LIN {X 0,Y 679.912,Z 1280.609,A -85,B 0,C 180,E1 32312.866,E2 32312.866} C_VEL
LIN {X 0,Y 679.874,Z 1281.737,A -85,B 0,C 180,E1 32311.011,E2 32311.011} C_VEL
LIN {X 0,Y 679.863,Z 1281.827,A -85,B 0,C 180,E1 32309.326,E2 32309.326} C_VEL
LIN {X 0,Y 679.905,Z 1280.946,A -85,B 0,C 180,E1 32307.556,E2 32307.556} C_VEL
LIN {X 0,Y 679.915,Z 1278.919,A -85,B 0,C 180,E1 32305.614,E2 32305.614} C_VEL
LIN {X 0,Y 679.929,Z 1274.906,A -85,B 0,C 180,E1 32303.329,E2 32303.329} C_VEL
LIN {X 0,Y 679.943,Z 1269.331,A -85,B 0,C 180,E1 32301.118,E2 32301.118} C_VEL
LIN {X 0,Y 680.017,Z 1263.356,A -85,B 0,C 180,E1 32299.238,E2 32299.238} C_VEL
LIN {X 0,Y 680.138,Z 1256.508,A -85,B 0,C 180,E1 32297.433,E2 32297.433} C_VEL
LIN {X 0,Y 680.303,Z 1248.399,A -85,B 0,C 180,E1 32295.6,E2 32295.6} C_VEL
LIN {X 0,Y 680.525,Z 1238.351,A -85,B 0,C 180,E1 32293.628,E2 32293.628} C_VEL
LIN {X 0,Y 680.966,Z 1224.744,A -85,B 0,C 180,E1 32291.331,E2 32291.331} C_VEL
LIN {X 0,Y 681.406,Z 1211.769,A -85,B 0,C 180,E1 32289.423,E2 32289.423} C_VEL
LIN {X 0,Y 681.969,Z 1198.553,A -85,B 0,C 180,E1 32287.683,E2 32287.683} C_VEL
LIN {X 0,Y 682.78,Z 1180.927,A -85,B 0,C 180,E1 32285.609,E2 32285.609} C_VEL
LIN {X 0,Y 683.632,Z 1163.822,A -85,B 0,C 180,E1 32283.831,E2 32283.831} C_VEL
LIN {X 0,Y 684.499,Z 1146.752,A -85,B 0,C 180,E1 32282.227,E2 32282.227} C_VEL
LIN {X 0,Y 685.785,Z 1124.203,A -85,B 0,C 180,E1 32280.341,E2 32280.341} C_VEL
LIN {X 0,Y 686.866,Z 1105.235,A -85,B 0,C 180,E1 32278.932,E2 32278.932} C_VEL
LIN {X 0,Y 687.97,Z 1085.493,A -85,B 0,C 180,E1 32277.61,E2 32277.61} C_VEL
LIN {X 0,Y 689.441,Z 1059.992,A -85,B 0,C 180,E1 32276.108,E2 32276.108} C_VEL
LIN {X 0,Y 690.593,Z 1038.701,A -85,B 0,C 180,E1 32275.016,E2 32275.016} C_VEL
LIN {X 0,Y 691.622,Z 1018.737,A -85,B 0,C 180,E1 32274.11,E2 32274.11} C_VEL
LIN {X 0,Y 692.593,Z 998.313,A -85,B 0,C 180,E1 32273.296,E2 32273.296} C_VEL
LIN {X 0,Y 693.528,Z 975.949,A -85,B 0,C 180,E1 32272.526,E2 32272.526} C_VEL
LIN {X 0,Y 694.563,Z 949.849,A -85,B 0,C 180,E1 32271.785,E2 32271.785} C_VEL
LIN {X 0,Y 695.355,Z 923.524,A -85,B 0,C 180,E1 32271.209,E2 32271.209} C_VEL
LIN {X 0,Y 695.921,Z 898.887,A -85,B 0,C 180,E1 32270.809,E2 32270.809} C_VEL
LIN {X 0,Y 698.303,Z 673.986,A -85,B 0,C 180,E1 32267.976,E2 32267.976} C_VEL
LIN {X 0,Y 700.559,Z 471.336,A -85,B 0,C 180,E1 32265.348,E2 32265.348} C_VEL
LIN {X 0,Y 700.664,Z 446.208,A -85,B 0,C 180,E1 32265,E2 32265} C_VEL
LIN {X 0,Y 696.356,Z 426.818,A -85,B 0,C 180,E1 32264.352,E2 32264.352} C_VEL
LIN {X 0,Y 698.129,Z 385.1,A -85,B 0,C 180,E1 32261.709,E2 32261.709} C_VEL
LIN {X 0,Y 698.689,Z 371.907,A -85,B 0,C 180,E1 32260.845,E2 32260.845} C_VEL
LIN {X 0,Y 684.161,Z 344.352,A -85,B 0,C 180,E1 32257.655,E2 32257.655} C_VEL
LIN {X 0,Y 682.069,Z 340.229,A -85,B 0,C 180,E1 32257.156,E2 32257.156} C_VEL
LIN {X 0,Y 680.532,Z 336.669,A -85,B 0,C 180,E1 32256.697,E2 32256.697} C_VEL
LIN {X 0,Y 680.502,Z 336.461,A -85,B 0,C 180,E1 32254.78,E2 32254.78} C_VEL
LIN {X 0,Y 680.517,Z 336.464,A -85,B 0,C 180,E1 32251.836,E2 32251.836} C_VEL
LIN {X 0,Y 680.507,Z 336.459,A -85,B 0,C 180,E1 32248.812,E2 32248.812} C_VEL
LIN {X 0,Y 680.521,Z 336.455,A -85,B 0,C 180,E1 32245.754,E2 32245.754} C_VEL
LIN {X 0,Y 680.506,Z 336.467,A -85,B 0,C 180,E1 32242.642,E2 32242.642} C_VEL
LIN {X 0,Y 680.523,Z 336.458,A -85,B 0,C 180,E1 32239.573,E2 32239.573} C_VEL
LIN {X 0,Y 680.505,Z 336.464,A -85,B 0,C 180,E1 32236.474,E2 32236.474} C_VEL
LIN {X 0,Y 680.526,Z 336.457,A -85,B 0,C 180,E1 32233.424,E2 32233.424} C_VEL
LIN {X 0,Y 680.505,Z 336.465,A -85,B 0,C 180,E1 32230.327,E2 32230.327} C_VEL
LIN {X 0,Y 680.526,Z 336.455,A -85,B 0,C 180,E1 32227.259,E2 32227.259} C_VEL
LIN {X 0,Y 680.502,Z 336.466,A -85,B 0,C 180,E1 32224.129,E2 32224.129} C_VEL
LIN {X 0,Y 680.518,Z 336.451,A -85,B 0,C 180,E1 32221.094,E2 32221.094} C_VEL
LIN {X 0,Y 680.501,Z 336.465,A -85,B 0,C 180,E1 32217.979,E2 32217.979} C_VEL
LIN {X 0,Y 680.509,Z 336.456,A -85,B 0,C 180,E1 32214.996,E2 32214.996} C_VEL
LIN {X 0,Y 680.499,Z 336.465,A -85,B 0,C 180,E1 32211.806,E2 32211.806} C_VEL
LIN {X 0,Y 680.497,Z 336.458,A -85,B 0,C 180,E1 32208.902,E2 32208.902} C_VEL
LIN {X 0,Y 680.505,Z 336.465,A -85,B 0,C 180,E1 32205.709,E2 32205.709} C_VEL
LIN {X 0,Y 680.486,Z 336.455,A -85,B 0,C 180,E1 32202.822,E2 32202.822} C_VEL
LIN {X 0,Y 680.522,Z 336.462,A -85,B 0,C 180,E1 32199.711,E2 32199.711} C_VEL
LIN {X 0,Y 680.475,Z 336.457,A -85,B 0,C 180,E1 32196.809,E2 32196.809} C_VEL
LIN {X 0,Y 680.527,Z 336.461,A -85,B 0,C 180,E1 32193.846,E2 32193.846} C_VEL
LIN {X 0,Y 680.473,Z 336.459,A -85,B 0,C 180,E1 32190.897,E2 32190.897} C_VEL
LIN {X 0,Y 680.524,Z 336.463,A -85,B 0,C 180,E1 32189.443,E2 32189.443} C_VEL
LIN {X 0,Y 679.498,Z 336.6,A -85,B 0,C 180,E1 32188.795,E2 32188.795} C_VEL
LIN {X 0,Y 673.053,Z 337.39,A -85,B 0,C 180,E1 32186.977,E2 32186.977} C_VEL
LIN {X 0,Y 672.532,Z 337.45,A -85,B 0,C 180,E1 32186.504,E2 32186.504} C_VEL
LIN {X 0,Y 672.587,Z 337.447,A -85,B 0,C 180,E1 32183.512,E2 32183.512} C_VEL
LIN {X 0,Y 672.53,Z 337.452,A -85,B 0,C 180,E1 32180.591,E2 32180.591} C_VEL
LIN {X 0,Y 672.563,Z 337.445,A -85,B 0,C 180,E1 32177.762,E2 32177.762} C_VEL
LIN {X 0,Y 672.544,Z 337.454,A -85,B 0,C 180,E1 32174.685,E2 32174.685} C_VEL
LIN {X 0,Y 672.526,Z 337.448,A -85,B 0,C 180,E1 32171.979,E2 32171.979} C_VEL
LIN {X 0,Y 672.59,Z 337.451,A -85,B 0,C 180,E1 32168.964,E2 32168.964} C_VEL
LIN {X 0,Y 672.519,Z 337.45,A -85,B 0,C 180,E1 32166.069,E2 32166.069} C_VEL
LIN {X 0,Y 672.562,Z 337.45,A -85,B 0,C 180,E1 32163.27,E2 32163.27} C_VEL
LIN {X 0,Y 672.53,Z 337.451,A -85,B 0,C 180,E1 32160.167,E2 32160.167} C_VEL
LIN {X 0,Y 672.519,Z 337.451,A -85,B 0,C 180,E1 32157.541,E2 32157.541} C_VEL
LIN {X 0,Y 672.585,Z 337.452,A -85,B 0,C 180,E1 32154.505,E2 32154.505} C_VEL
LIN {X 0,Y 672.512,Z 337.453,A -85,B 0,C 180,E1 32151.637,E2 32151.637} C_VEL
LIN {X 0,Y 672.545,Z 337.452,A -85,B 0,C 180,E1 32148.911,E2 32148.911} C_VEL
LIN {X 0,Y 672.525,Z 337.452,A -85,B 0,C 180,E1 32145.788,E2 32145.788} C_VEL
LIN {X 0,Y 672.505,Z 337.454,A -85,B 0,C 180,E1 32143.236,E2 32143.236} C_VEL
LIN {X 0,Y 672.566,Z 337.453,A -85,B 0,C 180,E1 32140.45,E2 32140.45} C_VEL
LIN {X 0,Y 672.511,Z 337.455,A -85,B 0,C 180,E1 32137.432,E2 32137.432} C_VEL
LIN {X 0,Y 672.501,Z 337.451,A -85,B 0,C 180,E1 32134.947,E2 32134.947} C_VEL
LIN {X 0,Y 672.58,Z 337.45,A -85,B 0,C 180,E1 32132.045,E2 32132.045} C_VEL
LIN {X 0,Y 672.505,Z 337.457,A -85,B 0,C 180,E1 32129.148,E2 32129.148} C_VEL
LIN {X 0,Y 672.498,Z 337.444,A -85,B 0,C 180,E1 32126.591,E2 32126.591} C_VEL
LIN {X 0,Y 672.576,Z 337.438,A -85,B 0,C 180,E1 32123.598,E2 32123.598} C_VEL
LIN {X 0,Y 672.493,Z 337.458,A -85,B 0,C 180,E1 32120.76,E2 32120.76} C_VEL
LIN {X 0,Y 672.498,Z 337.454,A -85,B 0,C 180,E1 32118.247,E2 32118.247} C_VEL
LIN {X 0,Y 672.554,Z 337.396,A -85,B 0,C 180,E1 32115.273,E2 32115.273} C_VEL
LIN {X 0,Y 672.486,Z 337.444,A -85,B 0,C 180,E1 32112.522,E2 32112.522} C_VEL
LIN {X 0,Y 672.557,Z 337.781,A -85,B 0,C 180,E1 32111.853,E2 32111.853} C_VEL
LIN {X 0,Y 673.067,Z 339.501,A -85,B 0,C 180,E1 32111.692,E2 32111.692} C_VEL
LIN {X 0,Y 675.158,Z 342.401,A -85,B 0,C 180,E1 32111.458,E2 32111.458} C_VEL
LIN {X 0,Y 676.417,Z 343.843,A -85,B 0,C 180,E1 32111.324,E2 32111.324} C_VEL
LIN {X 0,Y 679.051,Z 347.701,A -85,B 0,C 180,E1 32111.034,E2 32111.034} C_VEL
LIN {X 0,Y 690.723,Z 363.983,A -85,B 0,C 180,E1 32109.803,E2 32109.803} C_VEL
LIN {X 0,Y 694.272,Z 369.404,A -85,B 0,C 180,E1 32109.435,E2 32109.435} C_VEL
LIN {X 0,Y 691.631,Z 585.542,A -85,B 0,C 180,E1 32106.635,E2 32106.635} C_VEL
LIN {X 0,Y 689.568,Z 757.13,A -85,B 0,C 180,E1 32104.45,E2 32104.45} C_VEL
LIN {X 0,Y 688.782,Z 783.452,A -85,B 0,C 180,E1 32103.968,E2 32103.968} C_VEL
LIN {X 0,Y 687.772,Z 810.9,A -85,B 0,C 180,E1 32103.292,E2 32103.292} C_VEL
LIN {X 0,Y 686.614,Z 836.969,A -85,B 0,C 180,E1 32102.482,E2 32102.482} C_VEL
LIN {X 0,Y 685.243,Z 863.991,A -85,B 0,C 180,E1 32101.454,E2 32101.454} C_VEL
LIN {X 0,Y 683.973,Z 886.619,A -85,B 0,C 180,E1 32100.439,E2 32100.439} C_VEL
LIN {X 0,Y 682.54,Z 910.71,A -85,B 0,C 180,E1 32099.198,E2 32099.198} C_VEL
LIN {X 0,Y 680.907,Z 936.023,A -85,B 0,C 180,E1 32097.689,E2 32097.689} C_VEL
LIN {X 0,Y 679.643,Z 956.28,A -85,B 0,C 180,E1 32096.315,E2 32096.315} C_VEL
LIN {X 0,Y 678.282,Z 978.203,A -85,B 0,C 180,E1 32094.648,E2 32094.648} C_VEL
LIN {X 0,Y 676.938,Z 999.251,A -85,B 0,C 180,E1 32092.835,E2 32092.835} C_VEL
LIN {X 0,Y 675.887,Z 1017.79,A -85,B 0,C 180,E1 32091.044,E2 32091.044} C_VEL
LIN {X 0,Y 674.833,Z 1036.227,A -85,B 0,C 180,E1 32089.037,E2 32089.037} C_VEL
LIN {X 0,Y 674.017,Z 1053.07,A -85,B 0,C 180,E1 32086.969,E2 32086.969} C_VEL
LIN {X 0,Y 673.315,Z 1068.958,A -85,B 0,C 180,E1 32084.741,E2 32084.741} C_VEL
LIN {X 0,Y 672.867,Z 1081.301,A -85,B 0,C 180,E1 32082.771,E2 32082.771} C_VEL
LIN {X 0,Y 672.493,Z 1093.06,A -85,B 0,C 180,E1 32080.635,E2 32080.635} C_VEL
LIN {X 0,Y 672.222,Z 1104.249,A -85,B 0,C 180,E1 32078.227,E2 32078.227} C_VEL
LIN {X 0,Y 672.062,Z 1112.122,A -85,B 0,C 180,E1 32076.204,E2 32076.204} C_VEL
LIN {X 0,Y 671.984,Z 1118.828,A -85,B 0,C 180,E1 32074.123,E2 32074.123} C_VEL
LIN {X 0,Y 671.93,Z 1124.669,A -85,B 0,C 180,E1 32071.823,E2 32071.823} C_VEL
LIN {X 0,Y 671.911,Z 1128.607,A -85,B 0,C 180,E1 32069.608,E2 32069.608} C_VEL
LIN {X 0,Y 671.882,Z 1130.912,A -85,B 0,C 180,E1 32067.508,E2 32067.508} C_VEL
LIN {X 0,Y 671.901,Z 1131.864,A -85,B 0,C 180,E1 32065.567,E2 32065.567} C_VEL
LIN {X 0,Y 671.887,Z 1131.578,A -85,B 0,C 180,E1 32063.32,E2 32063.32} C_VEL
LIN {X 0,Y 671.909,Z 1129.575,A -85,B 0,C 180,E1 32061.017,E2 32061.017} C_VEL
LIN {X 0,Y 671.92,Z 1126.17,A -85,B 0,C 180,E1 32058.84,E2 32058.84} C_VEL
LIN {X 0,Y 671.953,Z 1120.892,A -85,B 0,C 180,E1 32056.512,E2 32056.512} C_VEL
LIN {X 0,Y 671.997,Z 1113.905,A -85,B 0,C 180,E1 32054.212,E2 32054.212} C_VEL
LIN {X 0,Y 672.161,Z 1106.347,A -85,B 0,C 180,E1 32052.195,E2 32052.195} C_VEL
LIN {X 0,Y 672.346,Z 1097.951,A -85,B 0,C 180,E1 32050.28,E2 32050.28} C_VEL
LIN {X 0,Y 672.66,Z 1086.935,A -85,B 0,C 180,E1 32048.118,E2 32048.118} C_VEL
LIN {X 0,Y 673.123,Z 1073.623,A -85,B 0,C 180,E1 32045.883,E2 32045.883} C_VEL
LIN {X 0,Y 673.696,Z 1060.257,A -85,B 0,C 180,E1 32043.915,E2 32043.915} C_VEL
LIN {X 0,Y 674.445,Z 1044.62,A -85,B 0,C 180,E1 32041.869,E2 32041.869} C_VEL
LIN {X 0,Y 675.363,Z 1026.896,A -85,B 0,C 180,E1 32039.83,E2 32039.83} C_VEL
LIN {X 0,Y 676.458,Z 1007.895,A -85,B 0,C 180,E1 32037.882,E2 32037.882} C_VEL
LIN {X 0,Y 677.675,Z 987.343,A -85,B 0,C 180,E1 32036.024,E2 32036.024} C_VEL
LIN {X 0,Y 678.875,Z 968.036,A -85,B 0,C 180,E1 32034.464,E2 32034.464} C_VEL
LIN {X 0,Y 680.414,Z 944.599,A -85,B 0,C 180,E1 32032.782,E2 32032.782} C_VEL
LIN {X 0,Y 681.858,Z 921.205,A -85,B 0,C 180,E1 32031.313,E2 32031.313} C_VEL
LIN {X 0,Y 683.375,Z 896.661,A -85,B 0,C 180,E1 32029.962,E2 32029.962} C_VEL
LIN {X 0,Y 684.813,Z 872.081,A -85,B 0,C 180,E1 32028.802,E2 32028.802} C_VEL
LIN {X 0,Y 686.072,Z 848.377,A -85,B 0,C 180,E1 32027.843,E2 32027.843} C_VEL
LIN {X 0,Y 687.209,Z 824.159,A -85,B 0,C 180,E1 32027.009,E2 32027.009} C_VEL
LIN {X 0,Y 688.249,Z 798.684,A -85,B 0,C 180,E1 32026.296,E2 32026.296} C_VEL
LIN {X 0,Y 689.148,Z 771.844,A -85,B 0,C 180,E1 32025.71,E2 32025.71} C_VEL
LIN {X 0,Y 689.804,Z 745.156,A -85,B 0,C 180,E1 32025.292,E2 32025.292} C_VEL
LIN {X 0,Y 692.457,Z 516.247,A -85,B 0,C 180,E1 32022.387,E2 32022.387} C_VEL
LIN {X 0,Y 694.14,Z 368.783,A -85,B 0,C 180,E1 32020.455,E2 32020.455} C_VEL
LIN {X 0,Y 682.65,Z 352.629,A -85,B 0,C 180,E1 32019.262,E2 32019.262} C_VEL
LIN {X 0,Y 678.852,Z 347.456,A -85,B 0,C 180,E1 32018.855,E2 32018.855} C_VEL
LIN {X 0,Y 676.214,Z 343.332,A -85,B 0,C 180,E1 32018.56,E2 32018.56} C_VEL
LIN {X 0,Y 673.433,Z 340.156,A -85,B 0,C 180,E1 32018.263,E2 32018.263} C_VEL
LIN {X 0,Y 672.641,Z 337.945,A -85,B 0,C 180,E1 32018.092,E2 32018.092} C_VEL
LIN {X 0,Y 672.533,Z 337.461,A -85,B 0,C 180,E1 32017.721,E2 32017.721} C_VEL
LIN {X 0,Y 672.565,Z 337.457,A -85,B 0,C 180,E1 32014.874,E2 32014.874} C_VEL
LIN {X 0,Y 672.558,Z 337.453,A -85,B 0,C 180,E1 32011.786,E2 32011.786} C_VEL
LIN {X 0,Y 672.567,Z 337.457,A -85,B 0,C 180,E1 32008.844,E2 32008.844} C_VEL
LIN {X 0,Y 672.574,Z 337.453,A -85,B 0,C 180,E1 32005.705,E2 32005.705} C_VEL
LIN {X 0,Y 672.609,Z 337.669,A -85,B 0,C 180,E1 32002.684,E2 32002.684} C_VEL
LIN {X 0,Y 673.551,Z 340.405,A -85,B 0,C 180,E1 32002.401,E2 32002.401} C_VEL
LIN {X 0,Y 681.915,Z 359.556,A -85,B 0,C 180,E1 32000.804,E2 32000.804} C_VEL
LIN {X 0,Y 692.135,Z 376.102,A -85,B 0,C 180,E1 31999.37,E2 31999.37} C_VEL
LIN {X 0,Y 692.068,Z 388.415,A -85,B 0,C 180,E1 31998.624,E2 31998.624} C_VEL
LIN {X 0,Y 690.346,Z 427.413,A -85,B 0,C 180,E1 31996.143,E2 31996.143} C_VEL
LIN {X 0,Y 695.134,Z 449.846,A -85,B 0,C 180,E1 31995.405,E2 31995.405} C_VEL
LIN {X 0,Y 692.574,Z 656.228,A -85,B 0,C 180,E1 31992.697,E2 31992.697} C_VEL
LIN {X 0,Y 689.978,Z 881.138,A -85,B 0,C 180,E1 31989.841,E2 31989.841} C_VEL
LIN {X 0,Y 689.357,Z 915.017,A -85,B 0,C 180,E1 31989.367,E2 31989.367} C_VEL
LIN {X 0,Y 688.525,Z 940.749,A -85,B 0,C 180,E1 31988.848,E2 31988.848} C_VEL
LIN {X 0,Y 687.58,Z 965.293,A -85,B 0,C 180,E1 31988.212,E2 31988.212} C_VEL
LIN {X 0,Y 686.32,Z 993.267,A -85,B 0,C 180,E1 31987.301,E2 31987.301} C_VEL
LIN {X 0,Y 685.156,Z 1015.348,A -85,B 0,C 180,E1 31986.438,E2 31986.438} C_VEL
LIN {X 0,Y 684.01,Z 1035.71,A -85,B 0,C 180,E1 31985.525,E2 31985.525} C_VEL
LIN {X 0,Y 682.83,Z 1055.546,A -85,B 0,C 180,E1 31984.52,E2 31984.52} C_VEL
LIN {X 0,Y 681.501,Z 1077.263,A -85,B 0,C 180,E1 31983.279,E2 31983.279} C_VEL
LIN {X 0,Y 679.886,Z 1101.91,A -85,B 0,C 180,E1 31981.67,E2 31981.67} C_VEL
LIN {X 0,Y 678.73,Z 1120.318,A -85,B 0,C 180,E1 31980.312,E2 31980.312} C_VEL
LIN {X 0,Y 677.63,Z 1138.267,A -85,B 0,C 180,E1 31978.849,E2 31978.849} C_VEL
LIN {X 0,Y 676.325,Z 1159.658,A -85,B 0,C 180,E1 31976.897,E2 31976.897} C_VEL
LIN {X 0,Y 675.387,Z 1175.867,A -85,B 0,C 180,E1 31975.234,E2 31975.234} C_VEL
LIN {X 0,Y 674.605,Z 1191.175,A -85,B 0,C 180,E1 31973.497,E2 31973.497} C_VEL
LIN {X 0,Y 673.761,Z 1208.709,A -85,B 0,C 180,E1 31971.254,E2 31971.254} C_VEL
LIN {X 0,Y 673.218,Z 1221.848,A -85,B 0,C 180,E1 31969.342,E2 31969.342} C_VEL
LIN {X 0,Y 672.774,Z 1233.631,A -85,B 0,C 180,E1 31967.416,E2 31967.416} C_VEL
LIN {X 0,Y 672.399,Z 1246.43,A -85,B 0,C 180,E1 31964.995,E2 31964.995} C_VEL
LIN {X 0,Y 672.194,Z 1255.439,A -85,B 0,C 180,E1 31962.98,E2 31962.98} C_VEL
LIN {X 0,Y 672.049,Z 1262.44,A -85,B 0,C 180,E1 31961.152,E2 31961.152} C_VEL
LIN {X 0,Y 671.943,Z 1268.053,A -85,B 0,C 180,E1 31959.421,E2 31959.421} C_VEL
LIN {X 0,Y 671.921,Z 1273.165,A -85,B 0,C 180,E1 31957.525,E2 31957.525} C_VEL
LIN {X 0,Y 671.914,Z 1277.634,A -85,B 0,C 180,E1 31955.294,E2 31955.294} C_VEL
LIN {X 0,Y 671.909,Z 1280.473,A -85,B 0,C 180,E1 31953.071,E2 31953.071} C_VEL
LIN {X 0,Y 671.881,Z 1281.715,A -85,B 0,C 180,E1 31951.108,E2 31951.108} C_VEL
LIN {X 0,Y 671.863,Z 1281.827,A -85,B 0,C 180,E1 31949.318,E2 31949.318} C_VEL
LIN {X 0,Y 671.906,Z 1280.946,A -85,B 0,C 180,E1 31947.527,E2 31947.527} C_VEL
LIN {X 0,Y 671.913,Z 1278.916,A -85,B 0,C 180,E1 31945.562,E2 31945.562} C_VEL
LIN {X 0,Y 671.928,Z 1274.907,A -85,B 0,C 180,E1 31943.249,E2 31943.249} C_VEL
LIN {X 0,Y 671.947,Z 1269.585,A -85,B 0,C 180,E1 31941.097,E2 31941.097} C_VEL
LIN {X 0,Y 672.032,Z 1263.357,A -85,B 0,C 180,E1 31939.108,E2 31939.108} C_VEL
LIN {X 0,Y 672.175,Z 1256.509,A -85,B 0,C 180,E1 31937.282,E2 31937.282} C_VEL
LIN {X 0,Y 672.367,Z 1248.072,A -85,B 0,C 180,E1 31935.356,E2 31935.356} C_VEL
LIN {X 0,Y 672.673,Z 1236.883,A -85,B 0,C 180,E1 31933.151,E2 31933.151} C_VEL
LIN {X 0,Y 673.15,Z 1223.595,A -85,B 0,C 180,E1 31930.926,E2 31930.926} C_VEL
LIN {X 0,Y 673.654,Z 1210.816,A -85,B 0,C 180,E1 31929.041,E2 31929.041} C_VEL
LIN {X 0,Y 674.368,Z 1195.631,A -85,B 0,C 180,E1 31927.038,E2 31927.038} C_VEL
LIN {X 0,Y 675.303,Z 1177.849,A -85,B 0,C 180,E1 31924.981,E2 31924.981} C_VEL
LIN {X 0,Y 676.174,Z 1161.986,A -85,B 0,C 180,E1 31923.334,E2 31923.334} C_VEL
LIN {X 0,Y 677.396,Z 1142.684,A -85,B 0,C 180,E1 31921.526,E2 31921.526} C_VEL
LIN {X 0,Y 678.65,Z 1121.656,A -85,B 0,C 180,E1 31919.792,E2 31919.792} C_VEL
LIN {X 0,Y 679.836,Z 1102.674,A -85,B 0,C 180,E1 31918.385,E2 31918.385} C_VEL
LIN {X 0,Y 681.412,Z 1078.863,A -85,B 0,C 180,E1 31916.816,E2 31916.816} C_VEL
LIN {X 0,Y 682.768,Z 1056.609,A -85,B 0,C 180,E1 31915.538,E2 31915.538} C_VEL
LIN {X 0,Y 683.963,Z 1036.588,A -85,B 0,C 180,E1 31914.517,E2 31914.517} C_VEL
LIN {X 0,Y 685.098,Z 1016.48,A -85,B 0,C 180,E1 31913.61,E2 31913.61} C_VEL
LIN {X 0,Y 686.225,Z 995.033,A -85,B 0,C 180,E1 31912.765,E2 31912.765} C_VEL
LIN {X 0,Y 687.499,Z 967.39,A -85,B 0,C 180,E1 31911.848,E2 31911.848} C_VEL
LIN {X 0,Y 688.481,Z 941.923,A -85,B 0,C 180,E1 31911.179,E2 31911.179} C_VEL
LIN {X 0,Y 689.293,Z 917.142,A -85,B 0,C 180,E1 31910.671,E2 31910.671} C_VEL
LIN {X 0,Y 689.928,Z 885.559,A -85,B 0,C 180,E1 31910.215,E2 31910.215} C_VEL
LIN {X 0,Y 692.512,Z 661.135,A -85,B 0,C 180,E1 31907.366,E2 31907.366} C_VEL
LIN {X 0,Y 695.041,Z 456.954,A -85,B 0,C 180,E1 31904.69,E2 31904.69} C_VEL
LIN {X 0,Y 694.977,Z 448.325,A -85,B 0,C 180,E1 31904.56,E2 31904.56} C_VEL
LIN {X 0,Y 690.269,Z 426.618,A -85,B 0,C 180,E1 31903.821,E2 31903.821} C_VEL
LIN {X 0,Y 692.248,Z 383.567,A -85,B 0,C 180,E1 31901.064,E2 31901.064} C_VEL
LIN {X 0,Y 692.335,Z 376.179,A -85,B 0,C 180,E1 31900.584,E2 31900.584} C_VEL
LIN {X 0,Y 678.51,Z 349.688,A -85,B 0,C 180,E1 31897.49,E2 31897.49} C_VEL
LIN {X 0,Y 676.416,Z 345.606,A -85,B 0,C 180,E1 31896.987,E2 31896.987} C_VEL
LIN {X 0,Y 673.968,Z 341.003,A -85,B 0,C 180,E1 31896.401,E2 31896.401} C_VEL
LIN {X 0,Y 672.605,Z 337.649,A -85,B 0,C 180,E1 31895.959,E2 31895.959} C_VEL
LIN {X 0,Y 672.572,Z 337.448,A -85,B 0,C 180,E1 31892.965,E2 31892.965} C_VEL
LIN {X 0,Y 672.584,Z 337.451,A -85,B 0,C 180,E1 31889.87,E2 31889.87} C_VEL
LIN {X 0,Y 672.569,Z 337.447,A -85,B 0,C 180,E1 31886.773,E2 31886.773} C_VEL
LIN {X 0,Y 672.582,Z 337.442,A -85,B 0,C 180,E1 31883.686,E2 31883.686} C_VEL
LIN {X 0,Y 672.571,Z 337.449,A -85,B 0,C 180,E1 31880.631,E2 31880.631} C_VEL
LIN {X 0,Y 672.585,Z 337.441,A -85,B 0,C 180,E1 31877.565,E2 31877.565} C_VEL
LIN {X 0,Y 672.568,Z 337.452,A -85,B 0,C 180,E1 31874.463,E2 31874.463} C_VEL
LIN {X 0,Y 672.58,Z 337.441,A -85,B 0,C 180,E1 31871.404,E2 31871.404} C_VEL
LIN {X 0,Y 672.568,Z 337.449,A -85,B 0,C 180,E1 31868.291,E2 31868.291} C_VEL
LIN {X 0,Y 672.575,Z 337.44,A -85,B 0,C 180,E1 31865.289,E2 31865.289} C_VEL
LIN {X 0,Y 672.566,Z 337.447,A -85,B 0,C 180,E1 31862.13,E2 31862.13} C_VEL
LIN {X 0,Y 672.569,Z 337.446,A -85,B 0,C 180,E1 31859.148,E2 31859.148} C_VEL
LIN {X 0,Y 672.568,Z 337.454,A -85,B 0,C 180,E1 31855.984,E2 31855.984} C_VEL
LIN {X 0,Y 672.563,Z 337.446,A -85,B 0,C 180,E1 31852.998,E2 31852.998} C_VEL
LIN {X 0,Y 672.566,Z 337.453,A -85,B 0,C 180,E1 31849.791,E2 31849.791} C_VEL
LIN {X 0,Y 672.557,Z 337.447,A -85,B 0,C 180,E1 31846.849,E2 31846.849} C_VEL
LIN {X 0,Y 672.57,Z 337.451,A -85,B 0,C 180,E1 31843.681,E2 31843.681} C_VEL
LIN {X 0,Y 672.55,Z 337.448,A -85,B 0,C 180,E1 31840.728,E2 31840.728} C_VEL
LIN {X 0,Y 672.582,Z 337.452,A -85,B 0,C 180,E1 31837.62,E2 31837.62} C_VEL
LIN {X 0,Y 672.538,Z 337.45,A -85,B 0,C 180,E1 31834.679,E2 31834.679} C_VEL
LIN {X 0,Y 672.59,Z 337.453,A -85,B 0,C 180,E1 31831.651,E2 31831.651} C_VEL
LIN {X 0,Y 672.532,Z 337.452,A -85,B 0,C 180,E1 31828.743,E2 31828.743} C_VEL
LIN {X 0,Y 672.532,Z 337.45,A -85,B 0,C 180,E1 31826.504,E2 31826.504} C_VEL
LIN {X 0,Y 671.563,Z 337.575,A -85,B 0,C 180,E1 31825.848,E2 31825.848} C_VEL
LIN {X 0,Y 665.179,Z 338.365,A -85,B 0,C 180,E1 31824.009,E2 31824.009} C_VEL
LIN {X 0,Y 664.648,Z 338.435,A -85,B 0,C 180,E1 31823.531,E2 31823.531} C_VEL
LIN {X 0,Y 664.591,Z 338.441,A -85,B 0,C 180,E1 31820.587,E2 31820.587} C_VEL
LIN {X 0,Y 664.627,Z 338.434,A -85,B 0,C 180,E1 31817.741,E2 31817.741} C_VEL
LIN {X 0,Y 664.601,Z 338.442,A -85,B 0,C 180,E1 31814.632,E2 31814.632} C_VEL
LIN {X 0,Y 664.594,Z 338.437,A -85,B 0,C 180,E1 31811.863,E2 31811.863} C_VEL
LIN {X 0,Y 664.629,Z 338.44,A -85,B 0,C 180,E1 31808.744,E2 31808.744} C_VEL
LIN {X 0,Y 664.58,Z 338.439,A -85,B 0,C 180,E1 31805.928,E2 31805.928} C_VEL
LIN {X 0,Y 664.65,Z 338.44,A -85,B 0,C 180,E1 31802.996,E2 31802.996} C_VEL
LIN {X 0,Y 664.584,Z 338.439,A -85,B 0,C 180,E1 31800.066,E2 31800.066} C_VEL
LIN {X 0,Y 664.586,Z 338.44,A -85,B 0,C 180,E1 31797.412,E2 31797.412} C_VEL
LIN {X 0,Y 664.625,Z 338.44,A -85,B 0,C 180,E1 31794.344,E2 31794.344} C_VEL
LIN {X 0,Y 664.573,Z 338.441,A -85,B 0,C 180,E1 31791.537,E2 31791.537} C_VEL
LIN {X 0,Y 664.634,Z 338.44,A -85,B 0,C 180,E1 31788.689,E2 31788.689} C_VEL
LIN {X 0,Y 664.576,Z 338.441,A -85,B 0,C 180,E1 31785.652,E2 31785.652} C_VEL
LIN {X 0,Y 664.569,Z 338.443,A -85,B 0,C 180,E1 31783.131,E2 31783.131} C_VEL
LIN {X 0,Y 664.645,Z 338.439,A -85,B 0,C 180,E1 31780.138,E2 31780.138} C_VEL
LIN {X 0,Y 664.564,Z 338.443,A -85,B 0,C 180,E1 31777.261,E2 31777.261} C_VEL
LIN {X 0,Y 664.57,Z 338.439,A -85,B 0,C 180,E1 31774.747,E2 31774.747} C_VEL
LIN {X 0,Y 664.622,Z 338.447,A -85,B 0,C 180,E1 31771.724,E2 31771.724} C_VEL
LIN {X 0,Y 664.559,Z 338.446,A -85,B 0,C 180,E1 31768.966,E2 31768.966} C_VEL
LIN {X 0,Y 664.582,Z 338.431,A -85,B 0,C 180,E1 31766.291,E2 31766.291} C_VEL
LIN {X 0,Y 664.569,Z 338.429,A -85,B 0,C 180,E1 31763.087,E2 31763.087} C_VEL
LIN {X 0,Y 664.554,Z 338.447,A -85,B 0,C 180,E1 31760.561,E2 31760.561} C_VEL
LIN {X 0,Y 664.615,Z 338.442,A -85,B 0,C 180,E1 31757.753,E2 31757.753} C_VEL
LIN {X 0,Y 664.55,Z 338.38,A -85,B 0,C 180,E1 31754.734,E2 31754.734} C_VEL
LIN {X 0,Y 664.572,Z 338.576,A -85,B 0,C 180,E1 31752.635,E2 31752.635} C_VEL
LIN {X 0,Y 664.766,Z 339.552,A -85,B 0,C 180,E1 31752.473,E2 31752.473} C_VEL
LIN {X 0,Y 666.632,Z 342.911,A -85,B 0,C 180,E1 31752.228,E2 31752.228} C_VEL
LIN {X 0,Y 668.544,Z 344.892,A -85,B 0,C 180,E1 31752.02,E2 31752.02} C_VEL
LIN {X 0,Y 671.321,Z 348.833,A -85,B 0,C 180,E1 31751.706,E2 31751.706} C_VEL
LIN {X 0,Y 686.131,Z 369.431,A -85,B 0,C 180,E1 31750.107,E2 31750.107} C_VEL
LIN {X 0,Y 688.505,Z 373.266,A -85,B 0,C 180,E1 31749.853,E2 31749.853} C_VEL
LIN {X 0,Y 685.594,Z 590.14,A -85,B 0,C 180,E1 31747.022,E2 31747.022} C_VEL
LIN {X 0,Y 683.386,Z 757.203,A -85,B 0,C 180,E1 31744.877,E2 31744.877} C_VEL
LIN {X 0,Y 682.543,Z 783.193,A -85,B 0,C 180,E1 31744.399,E2 31744.399} C_VEL
LIN {X 0,Y 681.444,Z 810.44,A -85,B 0,C 180,E1 31743.728,E2 31743.728} C_VEL
LIN {X 0,Y 680.187,Z 836.594,A -85,B 0,C 180,E1 31742.914,E2 31742.914} C_VEL
LIN {X 0,Y 678.655,Z 863.898,A -85,B 0,C 180,E1 31741.871,E2 31741.871} C_VEL
LIN {X 0,Y 677.262,Z 886.639,A -85,B 0,C 180,E1 31740.844,E2 31740.844} C_VEL
LIN {X 0,Y 675.702,Z 910.654,A -85,B 0,C 180,E1 31739.597,E2 31739.597} C_VEL
LIN {X 0,Y 673.965,Z 935.307,A -85,B 0,C 180,E1 31738.119,E2 31738.119} C_VEL
LIN {X 0,Y 672.487,Z 956.373,A -85,B 0,C 180,E1 31736.68,E2 31736.68} C_VEL
LIN {X 0,Y 670.995,Z 978.346,A -85,B 0,C 180,E1 31734.991,E2 31734.991} C_VEL
LIN {X 0,Y 669.526,Z 999.199,A -85,B 0,C 180,E1 31733.176,E2 31733.176} C_VEL
LIN {X 0,Y 668.336,Z 1017.912,A -85,B 0,C 180,E1 31731.349,E2 31731.349} C_VEL
LIN {X 0,Y 667.176,Z 1036.374,A -85,B 0,C 180,E1 31729.314,E2 31729.314} C_VEL
LIN {X 0,Y 666.266,Z 1053.277,A -85,B 0,C 180,E1 31727.211,E2 31727.211} C_VEL
LIN {X 0,Y 665.479,Z 1069.333,A -85,B 0,C 180,E1 31724.925,E2 31724.925} C_VEL
LIN {X 0,Y 664.988,Z 1081.264,A -85,B 0,C 180,E1 31722.996,E2 31722.996} C_VEL
LIN {X 0,Y 664.564,Z 1093.359,A -85,B 0,C 180,E1 31720.768,E2 31720.768} C_VEL
LIN {X 0,Y 664.258,Z 1104.408,A -85,B 0,C 180,E1 31718.35,E2 31718.35} C_VEL
LIN {X 0,Y 664.085,Z 1112.336,A -85,B 0,C 180,E1 31716.28,E2 31716.28} C_VEL
LIN {X 0,Y 663.992,Z 1119.01,A -85,B 0,C 180,E1 31714.173,E2 31714.173} C_VEL
LIN {X 0,Y 663.933,Z 1124.77,A -85,B 0,C 180,E1 31711.856,E2 31711.856} C_VEL
LIN {X 0,Y 663.912,Z 1128.694,A -85,B 0,C 180,E1 31709.603,E2 31709.603} C_VEL
LIN {X 0,Y 663.881,Z 1130.953,A -85,B 0,C 180,E1 31707.49,E2 31707.49} C_VEL
LIN {X 0,Y 663.899,Z 1131.882,A -85,B 0,C 180,E1 31705.515,E2 31705.515} C_VEL
LIN {X 0,Y 663.873,Z 1131.482,A -85,B 0,C 180,E1 31703.148,E2 31703.148} C_VEL
LIN {X 0,Y 663.914,Z 1129.4,A -85,B 0,C 180,E1 31700.82,E2 31700.82} C_VEL
LIN {X 0,Y 663.928,Z 1125.892,A -85,B 0,C 180,E1 31698.619,E2 31698.619} C_VEL
LIN {X 0,Y 663.974,Z 1120.5,A -85,B 0,C 180,E1 31696.266,E2 31696.266} C_VEL
LIN {X 0,Y 664.021,Z 1113.73,A -85,B 0,C 180,E1 31694.03,E2 31694.03} C_VEL
LIN {X 0,Y 664.215,Z 1106.149,A -85,B 0,C 180,E1 31691.99,E2 31691.99} C_VEL
LIN {X 0,Y 664.405,Z 1097.336,A -85,B 0,C 180,E1 31689.966,E2 31689.966} C_VEL
LIN {X 0,Y 664.825,Z 1085.753,A -85,B 0,C 180,E1 31687.692,E2 31687.692} C_VEL
LIN {X 0,Y 665.305,Z 1072.794,A -85,B 0,C 180,E1 31685.52,E2 31685.52} C_VEL
LIN {X 0,Y 665.947,Z 1059.362,A -85,B 0,C 180,E1 31683.529,E2 31683.529} C_VEL
LIN {X 0,Y 666.849,Z 1042.912,A -85,B 0,C 180,E1 31681.375,E2 31681.375} C_VEL
LIN {X 0,Y 667.826,Z 1025.756,A -85,B 0,C 180,E1 31679.4,E2 31679.4} C_VEL
LIN {X 0,Y 669.079,Z 1006.597,A -85,B 0,C 180,E1 31677.43,E2 31677.43} C_VEL
LIN {X 0,Y 670.423,Z 985.897,A -85,B 0,C 180,E1 31675.552,E2 31675.552} C_VEL
LIN {X 0,Y 671.932,Z 964.812,A -85,B 0,C 180,E1 31673.849,E2 31673.849} C_VEL
LIN {X 0,Y 673.56,Z 941.458,A -85,B 0,C 180,E1 31672.193,E2 31672.193} C_VEL
LIN {X 0,Y 675.134,Z 918.363,A -85,B 0,C 180,E1 31670.753,E2 31670.753} C_VEL
LIN {X 0,Y 676.891,Z 892.601,A -85,B 0,C 180,E1 31669.359,E2 31669.359} C_VEL
LIN {X 0,Y 678.313,Z 870.086,A -85,B 0,C 180,E1 31668.306,E2 31668.306} C_VEL
LIN {X 0,Y 679.63,Z 847.141,A -85,B 0,C 180,E1 31667.38,E2 31667.38} C_VEL
LIN {X 0,Y 680.944,Z 821.652,A -85,B 0,C 180,E1 31666.509,E2 31666.509} C_VEL
LIN {X 0,Y 682.069,Z 795.694,A -85,B 0,C 180,E1 31665.796,E2 31665.796} C_VEL
LIN {X 0,Y 683.027,Z 768.541,A -85,B 0,C 180,E1 31665.224,E2 31665.224} C_VEL
LIN {X 0,Y 683.712,Z 740.929,A -85,B 0,C 180,E1 31664.807,E2 31664.807} C_VEL
LIN {X 0,Y 686.62,Z 511.751,A -85,B 0,C 180,E1 31661.875,E2 31661.875} C_VEL
LIN {X 0,Y 688.421,Z 372.733,A -85,B 0,C 180,E1 31660.042,E2 31660.042} C_VEL
LIN {X 0,Y 678.252,Z 358.398,A -85,B 0,C 180,E1 31658.966,E2 31658.966} C_VEL
LIN {X 0,Y 671.209,Z 348.683,A -85,B 0,C 180,E1 31658.192,E2 31658.192} C_VEL
LIN {X 0,Y 668.47,Z 344.704,A -85,B 0,C 180,E1 31657.886,E2 31657.886} C_VEL
LIN {X 0,Y 665.442,Z 341.174,A -85,B 0,C 180,E1 31657.563,E2 31657.563} C_VEL
LIN {X 0,Y 664.706,Z 339.126,A -85,B 0,C 180,E1 31657.421,E2 31657.421} C_VEL
LIN {X 0,Y 664.6,Z 338.488,A -85,B 0,C 180,E1 31657.253,E2 31657.253} C_VEL
LIN {X 0,Y 664.646,Z 338.442,A -85,B 0,C 180,E1 31654.229,E2 31654.229} C_VEL
LIN {X 0,Y 664.603,Z 338.446,A -85,B 0,C 180,E1 31651.295,E2 31651.295} C_VEL
LIN {X 0,Y 664.645,Z 338.443,A -85,B 0,C 180,E1 31648.372,E2 31648.372} C_VEL
LIN {X 0,Y 664.615,Z 338.446,A -85,B 0,C 180,E1 31645.341,E2 31645.341} C_VEL
LIN {X 0,Y 664.656,Z 338.717,A -85,B 0,C 180,E1 31643.155,E2 31643.155} C_VEL
LIN {X 0,Y 668.289,Z 347.509,A -85,B 0,C 180,E1 31642.323,E2 31642.323} C_VEL
LIN {X 0,Y 675.542,Z 364.23,A -85,B 0,C 180,E1 31640.91,E2 31640.91} C_VEL
LIN {X 0,Y 685.154,Z 380.017,A -85,B 0,C 180,E1 31639.53,E2 31639.53} C_VEL
LIN {X 0,Y 685.545,Z 399.652,A -85,B 0,C 180,E1 31638.436,E2 31638.436} C_VEL
LIN {X 0,Y 684.326,Z 427.532,A -85,B 0,C 180,E1 31636.667,E2 31636.667} C_VEL
LIN {X 0,Y 689.481,Z 451.829,A -85,B 0,C 180,E1 31635.854,E2 31635.854} C_VEL
LIN {X 0,Y 686.669,Z 657.6,A -85,B 0,C 180,E1 31633.134,E2 31633.134} C_VEL
LIN {X 0,Y 683.822,Z 881.901,A -85,B 0,C 180,E1 31630.262,E2 31630.262} C_VEL
LIN {X 0,Y 683.128,Z 915.852,A -85,B 0,C 180,E1 31629.78,E2 31629.78} C_VEL
LIN {X 0,Y 682.235,Z 941.12,A -85,B 0,C 180,E1 31629.265,E2 31629.265} C_VEL
LIN {X 0,Y 681.212,Z 965.493,A -85,B 0,C 180,E1 31628.629,E2 31628.629} C_VEL
LIN {X 0,Y 679.832,Z 993.17,A -85,B 0,C 180,E1 31627.723,E2 31627.723} C_VEL
LIN {X 0,Y 678.556,Z 1015.344,A -85,B 0,C 180,E1 31626.85,E2 31626.85} C_VEL
LIN {X 0,Y 677.301,Z 1035.706,A -85,B 0,C 180,E1 31625.931,E2 31625.931} C_VEL
LIN {X 0,Y 675.954,Z 1056.439,A -85,B 0,C 180,E1 31624.87,E2 31624.87} C_VEL
LIN {X 0,Y 674.358,Z 1080.457,A -85,B 0,C 180,E1 31623.474,E2 31623.474} C_VEL
LIN {X 0,Y 672.684,Z 1103.243,A -85,B 0,C 180,E1 31621.948,E2 31621.948} C_VEL
LIN {X 0,Y 671.432,Z 1121.277,A -85,B 0,C 180,E1 31620.598,E2 31620.598} C_VEL
LIN {X 0,Y 670.12,Z 1141.036,A -85,B 0,C 180,E1 31618.959,E2 31618.959} C_VEL
LIN {X 0,Y 668.746,Z 1161.057,A -85,B 0,C 180,E1 31617.082,E2 31617.082} C_VEL
LIN {X 0,Y 667.744,Z 1176.695,A -85,B 0,C 180,E1 31615.452,E2 31615.452} C_VEL
LIN {X 0,Y 666.845,Z 1192.714,A -85,B 0,C 180,E1 31613.6,E2 31613.6} C_VEL
LIN {X 0,Y 665.942,Z 1209.529,A -85,B 0,C 180,E1 31611.398,E2 31611.398} C_VEL
LIN {X 0,Y 665.35,Z 1222.432,A -85,B 0,C 180,E1 31609.488,E2 31609.488} C_VEL
LIN {X 0,Y 664.855,Z 1234.344,A -85,B 0,C 180,E1 31607.504,E2 31607.504} C_VEL
LIN {X 0,Y 664.444,Z 1246.842,A -85,B 0,C 180,E1 31605.09,E2 31605.09} C_VEL
LIN {X 0,Y 664.217,Z 1255.797,A -85,B 0,C 180,E1 31603.05,E2 31603.05} C_VEL
LIN {X 0,Y 664.066,Z 1262.747,A -85,B 0,C 180,E1 31601.2,E2 31601.2} C_VEL
LIN {X 0,Y 663.951,Z 1268.31,A -85,B 0,C 180,E1 31599.448,E2 31599.448} C_VEL
LIN {X 0,Y 663.924,Z 1273.368,A -85,B 0,C 180,E1 31597.529,E2 31597.529} C_VEL
LIN {X 0,Y 663.917,Z 1277.928,A -85,B 0,C 180,E1 31595.184,E2 31595.184} C_VEL
LIN {X 0,Y 663.912,Z 1280.609,A -85,B 0,C 180,E1 31592.935,E2 31592.935} C_VEL
LIN {X 0,Y 663.876,Z 1281.737,A -85,B 0,C 180,E1 31591.036,E2 31591.036} C_VEL
LIN {X 0,Y 663.863,Z 1281.827,A -85,B 0,C 180,E1 31589.31,E2 31589.31} C_VEL
LIN {X 0,Y 663.906,Z 1280.947,A -85,B 0,C 180,E1 31587.497,E2 31587.497} C_VEL
LIN {X 0,Y 663.912,Z 1278.913,A -85,B 0,C 180,E1 31585.508,E2 31585.508} C_VEL
LIN {X 0,Y 663.932,Z 1274.907,A -85,B 0,C 180,E1 31583.167,E2 31583.167} C_VEL
LIN {X 0,Y 663.947,Z 1269.585,A -85,B 0,C 180,E1 31580.989,E2 31580.989} C_VEL
LIN {X 0,Y 664.051,Z 1263.357,A -85,B 0,C 180,E1 31578.976,E2 31578.976} C_VEL
LIN {X 0,Y 664.209,Z 1256.51,A -85,B 0,C 180,E1 31577.127,E2 31577.127} C_VEL
LIN {X 0,Y 664.423,Z 1248.073,A -85,B 0,C 180,E1 31575.177,E2 31575.177} C_VEL
LIN {X 0,Y 664.781,Z 1236.885,A -85,B 0,C 180,E1 31572.945,E2 31572.945} C_VEL
LIN {X 0,Y 665.306,Z 1223.594,A -85,B 0,C 180,E1 31570.693,E2 31570.693} C_VEL
LIN {X 0,Y 665.875,Z 1210.818,A -85,B 0,C 180,E1 31568.784,E2 31568.784} C_VEL
LIN {X 0,Y 666.714,Z 1195.004,A -85,B 0,C 180,E1 31566.676,E2 31566.676} C_VEL
LIN {X 0,Y 667.7,Z 1177.541,A -85,B 0,C 180,E1 31564.641,E2 31564.641} C_VEL
LIN {X 0,Y 668.711,Z 1161.521,A -85,B 0,C 180,E1 31562.964,E2 31562.964} C_VEL
LIN {X 0,Y 670.09,Z 1141.59,A -85,B 0,C 180,E1 31561.089,E2 31561.089} C_VEL
LIN {X 0,Y 671.431,Z 1121.28,A -85,B 0,C 180,E1 31559.402,E2 31559.402} C_VEL
LIN {X 0,Y 672.734,Z 1102.571,A -85,B 0,C 180,E1 31558.004,E2 31558.004} C_VEL
LIN {X 0,Y 674.461,Z 1078.811,A -85,B 0,C 180,E1 31556.426,E2 31556.426} C_VEL
LIN {X 0,Y 675.954,Z 1056.438,A -85,B 0,C 180,E1 31555.13,E2 31555.13} C_VEL
LIN {X 0,Y 677.301,Z 1035.708,A -85,B 0,C 180,E1 31554.069,E2 31554.069} C_VEL
LIN {X 0,Y 678.614,Z 1014.327,A -85,B 0,C 180,E1 31553.106,E2 31553.106} C_VEL
LIN {X 0,Y 680.103,Z 987.728,A -85,B 0,C 180,E1 31552.082,E2 31552.082} C_VEL
LIN {X 0,Y 681.346,Z 962.349,A -85,B 0,C 180,E1 31551.283,E2 31551.283} C_VEL
LIN {X 0,Y 682.343,Z 938.502,A -85,B 0,C 180,E1 31550.675,E2 31550.675} C_VEL
LIN {X 0,Y 683.271,Z 911.018,A -85,B 0,C 180,E1 31550.137,E2 31550.137} C_VEL
LIN {X 0,Y 684.018,Z 865.735,A -85,B 0,C 180,E1 31549.534,E2 31549.534} C_VEL
LIN {X 0,Y 686.885,Z 641.972,A -85,B 0,C 180,E1 31546.663,E2 31546.663} C_VEL
LIN {X 0,Y 689.457,Z 450.99,A -85,B 0,C 180,E1 31544.132,E2 31544.132} C_VEL
LIN {X 0,Y 684.229,Z 426.797,A -85,B 0,C 180,E1 31543.303,E2 31543.303} C_VEL
LIN {X 0,Y 685.827,Z 391.653,A -85,B 0,C 180,E1 31541.057,E2 31541.057} C_VEL
LIN {X 0,Y 686.041,Z 380.439,A -85,B 0,C 180,E1 31540.325,E2 31540.325} C_VEL
LIN {X 0,Y 672.868,Z 355.018,A -85,B 0,C 180,E1 31537.322,E2 31537.322} C_VEL
LIN {X 0,Y 668.349,Z 346.364,A -85,B 0,C 180,E1 31536.224,E2 31536.224} C_VEL
LIN {X 0,Y 666.326,Z 342.419,A -85,B 0,C 180,E1 31535.714,E2 31535.714} C_VEL
LIN {X 0,Y 664.698,Z 338.797,A -85,B 0,C 180,E1 31535.233,E2 31535.233} C_VEL
LIN {X 0,Y 664.629,Z 338.446,A -85,B 0,C 180,E1 31534.471,E2 31534.471} C_VEL
LIN {X 0,Y 664.639,Z 338.435,A -85,B 0,C 180,E1 31531.368,E2 31531.368} C_VEL
LIN {X 0,Y 664.624,Z 338.439,A -85,B 0,C 180,E1 31528.347,E2 31528.347} C_VEL
LIN {X 0,Y 664.637,Z 338.439,A -85,B 0,C 180,E1 31525.292,E2 31525.292} C_VEL
LIN {X 0,Y 664.617,Z 338.441,A -85,B 0,C 180,E1 31522.28,E2 31522.28} C_VEL
LIN {X 0,Y 664.638,Z 338.44,A -85,B 0,C 180,E1 31519.328,E2 31519.328} C_VEL
LIN {X 0,Y 664.618,Z 338.44,A -85,B 0,C 180,E1 31516.295,E2 31516.295} C_VEL
LIN {X 0,Y 664.644,Z 338.437,A -85,B 0,C 180,E1 31513.262,E2 31513.262} C_VEL
LIN {X 0,Y 664.621,Z 338.442,A -85,B 0,C 180,E1 31510.226,E2 31510.226} C_VEL
LIN {X 0,Y 664.649,Z 338.434,A -85,B 0,C 180,E1 31507.173,E2 31507.173} C_VEL
LIN {X 0,Y 664.62,Z 338.444,A -85,B 0,C 180,E1 31504.055,E2 31504.055} C_VEL
LIN {X 0,Y 664.645,Z 338.428,A -85,B 0,C 180,E1 31501.034,E2 31501.034} C_VEL
LIN {X 0,Y 664.62,Z 338.443,A -85,B 0,C 180,E1 31497.931,E2 31497.931} C_VEL
LIN {X 0,Y 664.639,Z 338.433,A -85,B 0,C 180,E1 31494.908,E2 31494.908} C_VEL
LIN {X 0,Y 664.621,Z 338.442,A -85,B 0,C 180,E1 31491.783,E2 31491.783} C_VEL
LIN {X 0,Y 664.631,Z 338.435,A -85,B 0,C 180,E1 31488.776,E2 31488.776} C_VEL
LIN {X 0,Y 664.62,Z 338.443,A -85,B 0,C 180,E1 31485.627,E2 31485.627} C_VEL
LIN {X 0,Y 664.62,Z 338.431,A -85,B 0,C 180,E1 31482.669,E2 31482.669} C_VEL
LIN {X 0,Y 664.623,Z 338.442,A -85,B 0,C 180,E1 31479.48,E2 31479.48} C_VEL
LIN {X 0,Y 664.609,Z 338.432,A -85,B 0,C 180,E1 31476.595,E2 31476.595} C_VEL
LIN {X 0,Y 664.637,Z 338.439,A -85,B 0,C 180,E1 31473.461,E2 31473.461} C_VEL
LIN {X 0,Y 664.596,Z 338.435,A -85,B 0,C 180,E1 31470.586,E2 31470.586} C_VEL
LIN {X 0,Y 664.649,Z 338.439,A -85,B 0,C 180,E1 31467.559,E2 31467.559} C_VEL
LIN {X 0,Y 664.591,Z 338.437,A -85,B 0,C 180,E1 31464.603,E2 31464.603} C_VEL
LIN {X 0,Y 664.648,Z 338.435,A -85,B 0,C 180,E1 31463.531,E2 31463.531} C_VEL
LIN {X 0,Y 663.655,Z 338.566,A -85,B 0,C 180,E1 31462.867,E2 31462.867} C_VEL
LIN {X 0,Y 657.196,Z 339.366,A -85,B 0,C 180,E1 31461.006,E2 31461.006} C_VEL
LIN {X 0,Y 656.651,Z 339.43,A -85,B 0,C 180,E1 31460.521,E2 31460.521} C_VEL
LIN {X 0,Y 656.703,Z 339.422,A -85,B 0,C 180,E1 31457.599,E2 31457.599} C_VEL
LIN {X 0,Y 656.657,Z 339.431,A -85,B 0,C 180,E1 31454.551,E2 31454.551} C_VEL
LIN {X 0,Y 656.664,Z 339.425,A -85,B 0,C 180,E1 31451.745,E2 31451.745} C_VEL
LIN {X 0,Y 656.664,Z 339.431,A -85,B 0,C 180,E1 31448.495,E2 31448.495} C_VEL
LIN {X 0,Y 656.649,Z 339.426,A -85,B 0,C 180,E1 31445.746,E2 31445.746} C_VEL
LIN {X 0,Y 656.697,Z 339.427,A -85,B 0,C 180,E1 31442.647,E2 31442.647} C_VEL
LIN {X 0,Y 656.639,Z 339.427,A -85,B 0,C 180,E1 31439.763,E2 31439.763} C_VEL
LIN {X 0,Y 656.71,Z 339.427,A -85,B 0,C 180,E1 31436.845,E2 31436.845} C_VEL
LIN {X 0,Y 656.638,Z 339.426,A -85,B 0,C 180,E1 31433.798,E2 31433.798} C_VEL
LIN {X 0,Y 656.649,Z 339.429,A -85,B 0,C 180,E1 31431.154,E2 31431.154} C_VEL
LIN {X 0,Y 656.665,Z 339.43,A -85,B 0,C 180,E1 31428.005,E2 31428.005} C_VEL
LIN {X 0,Y 656.63,Z 339.428,A -85,B 0,C 180,E1 31425.274,E2 31425.274} C_VEL
LIN {X 0,Y 656.704,Z 339.427,A -85,B 0,C 180,E1 31422.397,E2 31422.397} C_VEL
LIN {X 0,Y 656.63,Z 339.434,A -85,B 0,C 180,E1 31419.377,E2 31419.377} C_VEL
LIN {X 0,Y 656.633,Z 339.431,A -85,B 0,C 180,E1 31416.821,E2 31416.821} C_VEL
LIN {X 0,Y 656.679,Z 339.434,A -85,B 0,C 180,E1 31413.754,E2 31413.754} C_VEL
LIN {X 0,Y 656.621,Z 339.434,A -85,B 0,C 180,E1 31410.96,E2 31410.96} C_VEL
LIN {X 0,Y 656.646,Z 339.434,A -85,B 0,C 180,E1 31408.342,E2 31408.342} C_VEL
LIN {X 0,Y 656.638,Z 339.438,A -85,B 0,C 180,E1 31405.196,E2 31405.196} C_VEL
LIN {X 0,Y 656.613,Z 339.42,A -85,B 0,C 180,E1 31402.651,E2 31402.651} C_VEL
LIN {X 0,Y 656.649,Z 339.423,A -85,B 0,C 180,E1 31400.004,E2 31400.004} C_VEL
LIN {X 0,Y 656.627,Z 339.432,A -85,B 0,C 180,E1 31396.886,E2 31396.886} C_VEL
LIN {X 0,Y 656.601,Z 339.364,A -85,B 0,C 180,E1 31394.363,E2 31394.363} C_VEL
LIN {X 0,Y 656.726,Z 339.627,A -85,B 0,C 180,E1 31393.345,E2 31393.345} C_VEL
LIN {X 0,Y 657.058,Z 341.041,A -85,B 0,C 180,E1 31393.176,E2 31393.176} C_VEL
LIN {X 0,Y 659.005,Z 344.149,A -85,B 0,C 180,E1 31392.932,E2 31392.932} C_VEL
LIN {X 0,Y 660.572,Z 345.81,A -85,B 0,C 180,E1 31392.753,E2 31392.753} C_VEL
LIN {X 0,Y 663.118,Z 349.631,A -85,B 0,C 180,E1 31392.448,E2 31392.448} C_VEL
LIN {X 0,Y 664.813,Z 351.703,A -85,B 0,C 180,E1 31392.257,E2 31392.257} C_VEL
LIN {X 0,Y 679.754,Z 372.371,A -85,B 0,C 180,E1 31390.606,E2 31390.606} C_VEL
LIN {X 0,Y 682.774,Z 377.106,A -85,B 0,C 180,E1 31390.278,E2 31390.278} C_VEL
LIN {X 0,Y 679.588,Z 594.739,A -85,B 0,C 180,E1 31387.416,E2 31387.416} C_VEL
LIN {X 0,Y 677.24,Z 757.336,A -85,B 0,C 180,E1 31385.312,E2 31385.312} C_VEL
LIN {X 0,Y 676.33,Z 783.299,A -85,B 0,C 180,E1 31384.831,E2 31384.831} C_VEL
LIN {X 0,Y 675.132,Z 810.539,A -85,B 0,C 180,E1 31384.156,E2 31384.156} C_VEL
LIN {X 0,Y 673.785,Z 836.492,A -85,B 0,C 180,E1 31383.344,E2 31383.344} C_VEL
LIN {X 0,Y 672.082,Z 864.21,A -85,B 0,C 180,E1 31382.278,E2 31382.278} C_VEL
LIN {X 0,Y 670.52,Z 887.68,A -85,B 0,C 180,E1 31381.206,E2 31381.206} C_VEL
LIN {X 0,Y 668.818,Z 911.623,A -85,B 0,C 180,E1 31379.946,E2 31379.946} C_VEL
LIN {X 0,Y 667.018,Z 935.299,A -85,B 0,C 180,E1 31378.511,E2 31378.511} C_VEL
LIN {X 0,Y 665.353,Z 956.603,A -85,B 0,C 180,E1 31377.043,E2 31377.043} C_VEL
LIN {X 0,Y 663.728,Z 978.51,A -85,B 0,C 180,E1 31375.34,E2 31375.34} C_VEL
LIN {X 0,Y 662.12,Z 999.535,A -85,B 0,C 180,E1 31373.489,E2 31373.489} C_VEL
LIN {X 0,Y 660.735,Z 1019.199,A -85,B 0,C 180,E1 31371.541,E2 31371.541} C_VEL
LIN {X 0,Y 659.508,Z 1036.975,A -85,B 0,C 180,E1 31369.542,E2 31369.542} C_VEL
LIN {X 0,Y 658.512,Z 1053.708,A -85,B 0,C 180,E1 31367.428,E2 31367.428} C_VEL
LIN {X 0,Y 657.654,Z 1069.58,A -85,B 0,C 180,E1 31365.134,E2 31365.134} C_VEL
LIN {X 0,Y 657.095,Z 1081.655,A -85,B 0,C 180,E1 31363.152,E2 31363.152} C_VEL
LIN {X 0,Y 656.629,Z 1093.651,A -85,B 0,C 180,E1 31360.904,E2 31360.904} C_VEL
LIN {X 0,Y 656.299,Z 1104.291,A -85,B 0,C 180,E1 31358.545,E2 31358.545} C_VEL
LIN {X 0,Y 656.111,Z 1112.322,A -85,B 0,C 180,E1 31356.425,E2 31356.425} C_VEL
LIN {X 0,Y 656.001,Z 1119.191,A -85,B 0,C 180,E1 31354.225,E2 31354.225} C_VEL
LIN {X 0,Y 655.936,Z 1124.868,A -85,B 0,C 180,E1 31351.89,E2 31351.89} C_VEL
LIN {X 0,Y 655.912,Z 1128.781,A -85,B 0,C 180,E1 31349.598,E2 31349.598} C_VEL
LIN {X 0,Y 655.875,Z 1131.038,A -85,B 0,C 180,E1 31347.413,E2 31347.413} C_VEL
LIN {X 0,Y 655.9,Z 1131.939,A -85,B 0,C 180,E1 31345.268,E2 31345.268} C_VEL
LIN {X 0,Y 655.864,Z 1131.328,A -85,B 0,C 180,E1 31342.877,E2 31342.877} C_VEL
LIN {X 0,Y 655.917,Z 1129.209,A -85,B 0,C 180,E1 31340.614,E2 31340.614} C_VEL
LIN {X 0,Y 655.932,Z 1125.424,A -85,B 0,C 180,E1 31338.302,E2 31338.302} C_VEL
LIN {X 0,Y 655.977,Z 1120.111,A -85,B 0,C 180,E1 31336.015,E2 31336.015} C_VEL
LIN {X 0,Y 656.062,Z 1113.245,A -85,B 0,C 180,E1 31333.754,E2 31333.754} C_VEL
LIN {X 0,Y 656.26,Z 1105.599,A -85,B 0,C 180,E1 31331.692,E2 31331.692} C_VEL
LIN {X 0,Y 656.522,Z 1095.906,A -85,B 0,C 180,E1 31329.467,E2 31329.467} C_VEL
LIN {X 0,Y 657.003,Z 1083.496,A -85,B 0,C 180,E1 31327.081,E2 31327.081} C_VEL
LIN {X 0,Y 657.53,Z 1071.72,A -85,B 0,C 180,E1 31325.109,E2 31325.109} C_VEL
LIN {X 0,Y 658.298,Z 1057.223,A -85,B 0,C 180,E1 31322.96,E2 31322.96} C_VEL
LIN {X 0,Y 659.293,Z 1040.408,A -85,B 0,C 180,E1 31320.782,E2 31320.782} C_VEL
LIN {X 0,Y 660.344,Z 1024.611,A -85,B 0,C 180,E1 31318.959,E2 31318.959} C_VEL
LIN {X 0,Y 661.723,Z 1005.308,A -85,B 0,C 180,E1 31316.968,E2 31316.968} C_VEL
LIN {X 0,Y 663.252,Z 984.434,A -85,B 0,C 180,E1 31315.07,E2 31315.07} C_VEL
LIN {X 0,Y 664.944,Z 962.569,A -85,B 0,C 180,E1 31313.308,E2 31313.308} C_VEL
LIN {X 0,Y 666.628,Z 940.216,A -85,B 0,C 180,E1 31311.721,E2 31311.721} C_VEL
LIN {X 0,Y 668.344,Z 917.64,A -85,B 0,C 180,E1 31310.311,E2 31310.311} C_VEL
LIN {X 0,Y 670.194,Z 892.573,A -85,B 0,C 180,E1 31308.947,E2 31308.947} C_VEL
LIN {X 0,Y 671.738,Z 870.037,A -85,B 0,C 180,E1 31307.885,E2 31307.885} C_VEL
LIN {X 0,Y 673.167,Z 847.033,A -85,B 0,C 180,E1 31306.952,E2 31306.952} C_VEL
LIN {X 0,Y 674.613,Z 821.109,A -85,B 0,C 180,E1 31306.063,E2 31306.063} C_VEL
LIN {X 0,Y 675.838,Z 795.305,A -85,B 0,C 180,E1 31305.354,E2 31305.354} C_VEL
LIN {X 0,Y 676.858,Z 768.481,A -85,B 0,C 180,E1 31304.788,E2 31304.788} C_VEL
LIN {X 0,Y 677.594,Z 740.913,A -85,B 0,C 180,E1 31304.369,E2 31304.369} C_VEL
LIN {X 0,Y 680.771,Z 511.755,A -85,B 0,C 180,E1 31301.413,E2 31301.413} C_VEL
LIN {X 0,Y 682.671,Z 376.568,A -85,B 0,C 180,E1 31299.615,E2 31299.615} C_VEL
LIN {X 0,Y 670.9,Z 359.944,A -85,B 0,C 180,E1 31298.336,E2 31298.336} C_VEL
LIN {X 0,Y 666.386,Z 354.012,A -85,B 0,C 180,E1 31297.848,E2 31297.848} C_VEL
LIN {X 0,Y 663.353,Z 349.887,A -85,B 0,C 180,E1 31297.514,E2 31297.514} C_VEL
LIN {X 0,Y 660.548,Z 345.9,A -85,B 0,C 180,E1 31297.197,E2 31297.197} C_VEL
LIN {X 0,Y 659.491,Z 344.596,A -85,B 0,C 180,E1 31297.08,E2 31297.08} C_VEL
LIN {X 0,Y 657.31,Z 341.665,A -85,B 0,C 180,E1 31296.831,E2 31296.831} C_VEL
LIN {X 0,Y 656.785,Z 339.913,A -85,B 0,C 180,E1 31296.682,E2 31296.682} C_VEL
LIN {X 0,Y 656.712,Z 339.431,A -85,B 0,C 180,E1 31296.394,E2 31296.394} C_VEL
LIN {X 0,Y 656.66,Z 339.436,A -85,B 0,C 180,E1 31293.355,E2 31293.355} C_VEL
LIN {X 0,Y 656.708,Z 339.432,A -85,B 0,C 180,E1 31290.386,E2 31290.386} C_VEL
LIN {X 0,Y 656.673,Z 339.434,A -85,B 0,C 180,E1 31287.354,E2 31287.354} C_VEL
LIN {X 0,Y 656.704,Z 339.432,A -85,B 0,C 180,E1 31284.395,E2 31284.395} C_VEL
LIN {X 0,Y 656.746,Z 339.746,A -85,B 0,C 180,E1 31283.683,E2 31283.683} C_VEL
LIN {X 0,Y 659.176,Z 345.749,A -85,B 0,C 180,E1 31283.071,E2 31283.071} C_VEL
LIN {X 0,Y 665.182,Z 359.923,A -85,B 0,C 180,E1 31281.789,E2 31281.789} C_VEL
LIN {X 0,Y 669.691,Z 369.76,A -85,B 0,C 180,E1 31280.944,E2 31280.944} C_VEL
LIN {X 0,Y 678.143,Z 383.491,A -85,B 0,C 180,E1 31279.718,E2 31279.718} C_VEL
LIN {X 0,Y 678.762,Z 414.338,A -85,B 0,C 180,E1 31278.026,E2 31278.026} C_VEL
LIN {X 0,Y 678.352,Z 427.645,A -85,B 0,C 180,E1 31277.201,E2 31277.201} C_VEL
LIN {X 0,Y 683.871,Z 453.879,A -85,B 0,C 180,E1 31276.31,E2 31276.31} C_VEL
LIN {X 0,Y 680.807,Z 658.978,A -85,B 0,C 180,E1 31273.579,E2 31273.579} C_VEL
LIN {X 0,Y 677.69,Z 883.66,A -85,B 0,C 180,E1 31270.679,E2 31270.679} C_VEL
LIN {X 0,Y 676.925,Z 916.77,A -85,B 0,C 180,E1 31270.199,E2 31270.199} C_VEL
LIN {X 0,Y 675.988,Z 941.361,A -85,B 0,C 180,E1 31269.692,E2 31269.692} C_VEL
LIN {X 0,Y 674.892,Z 965.414,A -85,B 0,C 180,E1 31269.06,E2 31269.06} C_VEL
LIN {X 0,Y 673.376,Z 993.166,A -85,B 0,C 180,E1 31268.149,E2 31268.149} C_VEL
LIN {X 0,Y 671.949,Z 1016.053,A -85,B 0,C 180,E1 31267.24,E2 31267.24} C_VEL
LIN {X 0,Y 670.563,Z 1036.707,A -85,B 0,C 180,E1 31266.297,E2 31266.297} C_VEL
LIN {X 0,Y 669.029,Z 1058.5,A -85,B 0,C 180,E1 31265.163,E2 31265.163} C_VEL
LIN {X 0,Y 667.17,Z 1083.395,A -85,B 0,C 180,E1 31263.677,E2 31263.677} C_VEL
LIN {X 0,Y 665.527,Z 1104.238,A -85,B 0,C 180,E1 31262.257,E2 31262.257} C_VEL
LIN {X 0,Y 664.107,Z 1122.868,A -85,B 0,C 180,E1 31260.841,E2 31260.841} C_VEL
LIN {X 0,Y 662.506,Z 1144.723,A -85,B 0,C 180,E1 31258.977,E2 31258.977} C_VEL
LIN {X 0,Y 661.131,Z 1163.015,A -85,B 0,C 180,E1 31257.216,E2 31257.216} C_VEL
LIN {X 0,Y 660,Z 1179.495,A -85,B 0,C 180,E1 31255.453,E2 31255.453} C_VEL
LIN {X 0,Y 658.831,Z 1197.85,A -85,B 0,C 180,E1 31253.24,E2 31253.24} C_VEL
LIN {X 0,Y 658.048,Z 1211.799,A -85,B 0,C 180,E1 31251.339,E2 31251.339} C_VEL
LIN {X 0,Y 657.413,Z 1224.737,A -85,B 0,C 180,E1 31249.364,E2 31249.364} C_VEL
LIN {X 0,Y 656.812,Z 1238.281,A -85,B 0,C 180,E1 31246.995,E2 31246.995} C_VEL
LIN {X 0,Y 656.467,Z 1248.485,A -85,B 0,C 180,E1 31244.916,E2 31244.916} C_VEL
LIN {X 0,Y 656.235,Z 1256.871,A -85,B 0,C 180,E1 31242.943,E2 31242.943} C_VEL
LIN {X 0,Y 656.054,Z 1264.571,A -85,B 0,C 180,E1 31240.805,E2 31240.805} C_VEL
LIN {X 0,Y 655.963,Z 1271.914,A -85,B 0,C 180,E1 31238.238,E2 31238.238} C_VEL
LIN {X 0,Y 655.93,Z 1276.569,A -85,B 0,C 180,E1 31236.038,E2 31236.038} C_VEL
LIN {X 0,Y 655.914,Z 1279.993,A -85,B 0,C 180,E1 31233.671,E2 31233.671} C_VEL
LIN {X 0,Y 655.9,Z 1281.669,A -85,B 0,C 180,E1 31231.31,E2 31231.31} C_VEL
LIN {X 0,Y 655.864,Z 1281.849,A -85,B 0,C 180,E1 31229.389,E2 31229.389} C_VEL
LIN {X 0,Y 655.907,Z 1281.014,A -85,B 0,C 180,E1 31227.554,E2 31227.554} C_VEL
LIN {X 0,Y 655.914,Z 1279.024,A -85,B 0,C 180,E1 31225.541,E2 31225.541} C_VEL
LIN {X 0,Y 655.932,Z 1275.25,A -85,B 0,C 180,E1 31223.259,E2 31223.259} C_VEL
LIN {X 0,Y 655.953,Z 1269.839,A -85,B 0,C 180,E1 31220.967,E2 31220.967} C_VEL
LIN {X 0,Y 656.074,Z 1263.358,A -85,B 0,C 180,E1 31218.84,E2 31218.84} C_VEL
LIN {X 0,Y 656.239,Z 1256.511,A -85,B 0,C 180,E1 31216.968,E2 31216.968} C_VEL
LIN {X 0,Y 656.476,Z 1248.074,A -85,B 0,C 180,E1 31214.994,E2 31214.994} C_VEL
LIN {X 0,Y 656.889,Z 1236.886,A -85,B 0,C 180,E1 31212.733,E2 31212.733} C_VEL
LIN {X 0,Y 657.463,Z 1223.592,A -85,B 0,C 180,E1 31210.453,E2 31210.453} C_VEL
LIN {X 0,Y 658.102,Z 1210.82,A -85,B 0,C 180,E1 31208.521,E2 31208.521} C_VEL
LIN {X 0,Y 659.036,Z 1195.006,A -85,B 0,C 180,E1 31206.388,E2 31206.388} C_VEL
LIN {X 0,Y 660.114,Z 1177.504,A -85,B 0,C 180,E1 31204.325,E2 31204.325} C_VEL
LIN {X 0,Y 661.25,Z 1161.522,A -85,B 0,C 180,E1 31202.634,E2 31202.634} C_VEL
LIN {X 0,Y 662.74,Z 1141.59,A -85,B 0,C 180,E1 31200.737,E2 31200.737} C_VEL
LIN {X 0,Y 664.191,Z 1121.719,A -85,B 0,C 180,E1 31199.068,E2 31199.068} C_VEL
LIN {X 0,Y 665.611,Z 1103.236,A -85,B 0,C 180,E1 31197.671,E2 31197.671} C_VEL
LIN {X 0,Y 667.425,Z 1080.447,A -85,B 0,C 180,E1 31196.131,E2 31196.131} C_VEL
LIN {X 0,Y 669.161,Z 1056.441,A -85,B 0,C 180,E1 31194.724,E2 31194.724} C_VEL
LIN {X 0,Y 670.628,Z 1035.704,A -85,B 0,C 180,E1 31193.654,E2 31193.654} C_VEL
LIN {X 0,Y 672.135,Z 1013.08,A -85,B 0,C 180,E1 31192.631,E2 31192.631} C_VEL
LIN {X 0,Y 673.794,Z 985.655,A -85,B 0,C 180,E1 31191.586,E2 31191.586} C_VEL
LIN {X 0,Y 675.053,Z 961.899,A -85,B 0,C 180,E1 31190.84,E2 31190.84} C_VEL
LIN {X 0,Y 676.127,Z 938.103,A -85,B 0,C 180,E1 31190.232,E2 31190.232} C_VEL
LIN {X 0,Y 677.135,Z 910.424,A -85,B 0,C 180,E1 31189.692,E2 31189.692} C_VEL
LIN {X 0,Y 677.968,Z 862.65,A -85,B 0,C 180,E1 31189.054,E2 31189.054} C_VEL
LIN {X 0,Y 681.096,Z 639.504,A -85,B 0,C 180,E1 31186.166,E2 31186.166} C_VEL
LIN {X 0,Y 683.856,Z 453.075,A -85,B 0,C 180,E1 31183.677,E2 31183.677} C_VEL
LIN {X 0,Y 678.236,Z 426.786,A -85,B 0,C 180,E1 31182.763,E2 31182.763} C_VEL
LIN {X 0,Y 679.936,Z 385.345,A -85,B 0,C 180,E1 31180.121,E2 31180.121} C_VEL
LIN {X 0,Y 669.692,Z 365.14,A -85,B 0,C 180,E1 31177.746,E2 31177.746} C_VEL
LIN {X 0,Y 663.107,Z 352.314,A -85,B 0,C 180,E1 31176.128,E2 31176.128} C_VEL
LIN {X 0,Y 660.712,Z 347.824,A -85,B 0,C 180,E1 31175.53,E2 31175.53} C_VEL
LIN {X 0,Y 658.362,Z 343.395,A -85,B 0,C 180,E1 31174.93,E2 31174.93} C_VEL
LIN {X 0,Y 656.753,Z 339.843,A -85,B 0,C 180,E1 31174.444,E2 31174.444} C_VEL
LIN {X 0,Y 656.695,Z 339.423,A -85,B 0,C 180,E1 31173.763,E2 31173.763} C_VEL
LIN {X 0,Y 656.687,Z 339.425,A -85,B 0,C 180,E1 31170.771,E2 31170.771} C_VEL
LIN {X 0,Y 656.705,Z 339.427,A -85,B 0,C 180,E1 31167.769,E2 31167.769} C_VEL
LIN {X 0,Y 656.686,Z 339.428,A -85,B 0,C 180,E1 31164.633,E2 31164.633} C_VEL
LIN {X 0,Y 656.707,Z 339.426,A -85,B 0,C 180,E1 31161.621,E2 31161.621} C_VEL
LIN {X 0,Y 656.685,Z 339.423,A -85,B 0,C 180,E1 31158.464,E2 31158.464} C_VEL
LIN {X 0,Y 656.705,Z 339.423,A -85,B 0,C 180,E1 31155.363,E2 31155.363} C_VEL
LIN {X 0,Y 656.683,Z 339.423,A -85,B 0,C 180,E1 31152.308,E2 31152.308} C_VEL
LIN {X 0,Y 656.706,Z 339.423,A -85,B 0,C 180,E1 31149.288,E2 31149.288} C_VEL
LIN {X 0,Y 656.682,Z 339.425,A -85,B 0,C 180,E1 31146.137,E2 31146.137} C_VEL
LIN {X 0,Y 656.705,Z 339.425,A -85,B 0,C 180,E1 31143.055,E2 31143.055} C_VEL
LIN {X 0,Y 656.678,Z 339.431,A -85,B 0,C 180,E1 31139.913,E2 31139.913} C_VEL
LIN {X 0,Y 656.705,Z 339.423,A -85,B 0,C 180,E1 31136.858,E2 31136.858} C_VEL
LIN {X 0,Y 656.673,Z 339.43,A -85,B 0,C 180,E1 31133.706,E2 31133.706} C_VEL
LIN {X 0,Y 656.703,Z 339.423,A -85,B 0,C 180,E1 31130.712,E2 31130.712} C_VEL
LIN {X 0,Y 656.677,Z 339.431,A -85,B 0,C 180,E1 31127.602,E2 31127.602} C_VEL
LIN {X 0,Y 656.69,Z 339.425,A -85,B 0,C 180,E1 31124.637,E2 31124.637} C_VEL
LIN {X 0,Y 656.676,Z 339.432,A -85,B 0,C 180,E1 31121.444,E2 31121.444} C_VEL
LIN {X 0,Y 656.688,Z 339.425,A -85,B 0,C 180,E1 31118.472,E2 31118.472} C_VEL
LIN {X 0,Y 656.68,Z 339.433,A -85,B 0,C 180,E1 31115.342,E2 31115.342} C_VEL
LIN {X 0,Y 656.67,Z 339.427,A -85,B 0,C 180,E1 31112.426,E2 31112.426} C_VEL
LIN {X 0,Y 656.687,Z 339.433,A -85,B 0,C 180,E1 31109.229,E2 31109.229} C_VEL
LIN {X 0,Y 656.661,Z 339.427,A -85,B 0,C 180,E1 31106.34,E2 31106.34} C_VEL
LIN {X 0,Y 656.699,Z 339.431,A -85,B 0,C 180,E1 31103.214,E2 31103.214} C_VEL
LIN {X 0,Y 656.651,Z 339.43,A -85,B 0,C 180,E1 31100.521,E2 31100.521} C_VEL
LIN {X 0,Y 655.654,Z 339.554,A -85,B 0,C 180,E1 31099.849,E2 31099.849} C_VEL
LIN {X 0,Y 649.278,Z 340.347,A -85,B 0,C 180,E1 31097.965,E2 31097.965} C_VEL
LIN {X 0,Y 648.77,Z 340.411,A -85,B 0,C 180,E1 31097.475,E2 31097.475} C_VEL
LIN {X 0,Y 648.712,Z 340.419,A -85,B 0,C 180,E1 31094.408,E2 31094.408} C_VEL
LIN {X 0,Y 648.754,Z 340.412,A -85,B 0,C 180,E1 31091.492,E2 31091.492} C_VEL
LIN {X 0,Y 648.717,Z 340.42,A -85,B 0,C 180,E1 31088.4,E2 31088.4} C_VEL
LIN {X 0,Y 648.716,Z 340.415,A -85,B 0,C 180,E1 31085.635,E2 31085.635} C_VEL
LIN {X 0,Y 648.732,Z 340.418,A -85,B 0,C 180,E1 31082.436,E2 31082.436} C_VEL
LIN {X 0,Y 648.701,Z 340.415,A -85,B 0,C 180,E1 31079.655,E2 31079.655} C_VEL
LIN {X 0,Y 648.772,Z 340.414,A -85,B 0,C 180,E1 31076.632,E2 31076.632} C_VEL
LIN {X 0,Y 648.697,Z 340.414,A -85,B 0,C 180,E1 31073.711,E2 31073.711} C_VEL
LIN {X 0,Y 648.731,Z 340.417,A -85,B 0,C 180,E1 31070.951,E2 31070.951} C_VEL
LIN {X 0,Y 648.704,Z 340.421,A -85,B 0,C 180,E1 31067.769,E2 31067.769} C_VEL
LIN {X 0,Y 648.698,Z 340.416,A -85,B 0,C 180,E1 31065.099,E2 31065.099} C_VEL
LIN {X 0,Y 648.759,Z 340.417,A -85,B 0,C 180,E1 31062.099,E2 31062.099} C_VEL
LIN {X 0,Y 648.687,Z 340.423,A -85,B 0,C 180,E1 31059.225,E2 31059.225} C_VEL
LIN {X 0,Y 648.717,Z 340.419,A -85,B 0,C 180,E1 31056.549,E2 31056.549} C_VEL
LIN {X 0,Y 648.697,Z 340.422,A -85,B 0,C 180,E1 31053.358,E2 31053.358} C_VEL
LIN {X 0,Y 648.686,Z 340.423,A -85,B 0,C 180,E1 31050.707,E2 31050.707} C_VEL
LIN {X 0,Y 648.754,Z 340.401,A -85,B 0,C 180,E1 31047.703,E2 31047.703} C_VEL
LIN {X 0,Y 648.679,Z 340.426,A -85,B 0,C 180,E1 31044.782,E2 31044.782} C_VEL
LIN {X 0,Y 648.707,Z 340.41,A -85,B 0,C 180,E1 31042.115,E2 31042.115} C_VEL
LIN {X 0,Y 648.691,Z 340.405,A -85,B 0,C 180,E1 31038.981,E2 31038.981} C_VEL
LIN {X 0,Y 648.669,Z 340.395,A -85,B 0,C 180,E1 31036.45,E2 31036.45} C_VEL
LIN {X 0,Y 648.698,Z 340.552,A -85,B 0,C 180,E1 31034.153,E2 31034.153} C_VEL
LIN {X 0,Y 649.056,Z 341.962,A -85,B 0,C 180,E1 31033.959,E2 31033.959} C_VEL
LIN {X 0,Y 650.922,Z 344.95,A -85,B 0,C 180,E1 31033.715,E2 31033.715} C_VEL
LIN {X 0,Y 652.751,Z 346.774,A -85,B 0,C 180,E1 31033.501,E2 31033.501} C_VEL
LIN {X 0,Y 655.394,Z 350.736,A -85,B 0,C 180,E1 31033.173,E2 31033.173} C_VEL
LIN {X 0,Y 656.955,Z 352.787,A -85,B 0,C 180,E1 31032.986,E2 31032.986} C_VEL
LIN {X 0,Y 668.034,Z 367.783,A -85,B 0,C 180,E1 31031.714,E2 31031.714} C_VEL
LIN {X 0,Y 677.086,Z 380.645,A -85,B 0,C 180,E1 31030.714,E2 31030.714} C_VEL
LIN {X 0,Y 673.625,Z 598.467,A -85,B 0,C 180,E1 31027.829,E2 31027.829} C_VEL
LIN {X 0,Y 671.139,Z 757.296,A -85,B 0,C 180,E1 31025.757,E2 31025.757} C_VEL
LIN {X 0,Y 670.153,Z 783.463,A -85,B 0,C 180,E1 31025.269,E2 31025.269} C_VEL
LIN {X 0,Y 668.856,Z 810.679,A -85,B 0,C 180,E1 31024.591,E2 31024.591} C_VEL
LIN {X 0,Y 667.402,Z 836.676,A -85,B 0,C 180,E1 31023.771,E2 31023.771} C_VEL
LIN {X 0,Y 665.613,Z 863.658,A -85,B 0,C 180,E1 31022.731,E2 31022.731} C_VEL
LIN {X 0,Y 663.876,Z 887.671,A -85,B 0,C 180,E1 31021.629,E2 31021.629} C_VEL
LIN {X 0,Y 662.036,Z 911.658,A -85,B 0,C 180,E1 31020.355,E2 31020.355} C_VEL
LIN {X 0,Y 660.085,Z 935.46,A -85,B 0,C 180,E1 31018.9,E2 31018.9} C_VEL
LIN {X 0,Y 658.276,Z 956.66,A -85,B 0,C 180,E1 31017.426,E2 31017.426} C_VEL
LIN {X 0,Y 656.436,Z 979.256,A -85,B 0,C 180,E1 31015.648,E2 31015.648} C_VEL
LIN {X 0,Y 654.679,Z 1000.513,A -85,B 0,C 180,E1 31013.747,E2 31013.747} C_VEL
LIN {X 0,Y 653.138,Z 1020.265,A -85,B 0,C 180,E1 31011.754,E2 31011.754} C_VEL
LIN {X 0,Y 651.852,Z 1037.576,A -85,B 0,C 180,E1 31009.777,E2 31009.777} C_VEL
LIN {X 0,Y 650.767,Z 1054.138,A -85,B 0,C 180,E1 31007.651,E2 31007.651} C_VEL
LIN {X 0,Y 649.849,Z 1069.608,A -85,B 0,C 180,E1 31005.383,E2 31005.383} C_VEL
LIN {X 0,Y 649.219,Z 1081.719,A -85,B 0,C 180,E1 31003.37,E2 31003.37} C_VEL
LIN {X 0,Y 648.703,Z 1093.376,A -85,B 0,C 180,E1 31001.16,E2 31001.16} C_VEL
LIN {X 0,Y 648.337,Z 1104.325,A -85,B 0,C 180,E1 30998.707,E2 30998.707} C_VEL
LIN {X 0,Y 648.13,Z 1112.391,A -85,B 0,C 180,E1 30996.548,E2 30996.548} C_VEL
LIN {X 0,Y 648.008,Z 1119.371,A -85,B 0,C 180,E1 30994.278,E2 30994.278} C_VEL
LIN {X 0,Y 647.939,Z 1124.966,A -85,B 0,C 180,E1 30991.925,E2 30991.925} C_VEL
LIN {X 0,Y 647.913,Z 1128.868,A -85,B 0,C 180,E1 30989.593,E2 30989.593} C_VEL
LIN {X 0,Y 647.873,Z 1131.088,A -85,B 0,C 180,E1 30987.382,E2 30987.382} C_VEL
LIN {X 0,Y 647.906,Z 1131.972,A -85,B 0,C 180,E1 30985.113,E2 30985.113} C_VEL
LIN {X 0,Y 647.863,Z 1131.29,A -85,B 0,C 180,E1 30982.792,E2 30982.792} C_VEL
LIN {X 0,Y 647.917,Z 1129.265,A -85,B 0,C 180,E1 30980.601,E2 30980.601} C_VEL
LIN {X 0,Y 647.934,Z 1125.495,A -85,B 0,C 180,E1 30978.256,E2 30978.256} C_VEL
LIN {X 0,Y 647.987,Z 1119.966,A -85,B 0,C 180,E1 30975.85,E2 30975.85} C_VEL
LIN {X 0,Y 648.103,Z 1113.07,A -85,B 0,C 180,E1 30973.563,E2 30973.563} C_VEL
LIN {X 0,Y 648.293,Z 1105.762,A -85,B 0,C 180,E1 30971.567,E2 30971.567} C_VEL
LIN {X 0,Y 648.579,Z 1096.366,A -85,B 0,C 180,E1 30969.374,E2 30969.374} C_VEL
LIN {X 0,Y 649.094,Z 1084.253,A -85,B 0,C 180,E1 30966.99,E2 30966.99} C_VEL
LIN {X 0,Y 649.719,Z 1071.693,A -85,B 0,C 180,E1 30964.856,E2 30964.856} C_VEL
LIN {X 0,Y 650.577,Z 1056.92,A -85,B 0,C 180,E1 30962.643,E2 30962.643} C_VEL
LIN {X 0,Y 651.664,Z 1040.078,A -85,B 0,C 180,E1 30960.44,E2 30960.44} C_VEL
LIN {X 0,Y 652.84,Z 1024.252,A -85,B 0,C 180,E1 30958.596,E2 30958.596} C_VEL
LIN {X 0,Y 654.333,Z 1004.908,A -85,B 0,C 180,E1 30956.583,E2 30956.583} C_VEL
LIN {X 0,Y 655.987,Z 984.478,A -85,B 0,C 180,E1 30954.709,E2 30954.709} C_VEL
LIN {X 0,Y 657.824,Z 962.607,A -85,B 0,C 180,E1 30952.928,E2 30952.928} C_VEL
LIN {X 0,Y 659.663,Z 940.25,A -85,B 0,C 180,E1 30951.326,E2 30951.326} C_VEL
LIN {X 0,Y 661.537,Z 917.638,A -85,B 0,C 180,E1 30949.902,E2 30949.902} C_VEL
LIN {X 0,Y 663.529,Z 892.547,A -85,B 0,C 180,E1 30948.526,E2 30948.526} C_VEL
LIN {X 0,Y 665.261,Z 869.021,A -85,B 0,C 180,E1 30947.412,E2 30947.412} C_VEL
LIN {X 0,Y 666.878,Z 844.67,A -85,B 0,C 180,E1 30946.429,E2 30946.429} C_VEL
LIN {X 0,Y 668.525,Z 816.953,A -85,B 0,C 180,E1 30945.502,E2 30945.502} C_VEL
LIN {X 0,Y 669.85,Z 791.065,A -85,B 0,C 180,E1 30944.81,E2 30944.81} C_VEL
LIN {X 0,Y 670.847,Z 764.856,A -85,B 0,C 180,E1 30944.28,E2 30944.28} C_VEL
LIN {X 0,Y 671.656,Z 731.015,A -85,B 0,C 180,E1 30943.796,E2 30943.796} C_VEL
LIN {X 0,Y 675.096,Z 503.747,A -85,B 0,C 180,E1 30940.837,E2 30940.837} C_VEL
LIN {X 0,Y 676.981,Z 380.297,A -85,B 0,C 180,E1 30939.182,E2 30939.182} C_VEL
LIN {X 0,Y 663.135,Z 361.156,A -85,B 0,C 180,E1 30937.673,E2 30937.673} C_VEL
LIN {X 0,Y 656.37,Z 352.007,A -85,B 0,C 180,E1 30936.912,E2 30936.912} C_VEL
LIN {X 0,Y 652.922,Z 347.28,A -85,B 0,C 180,E1 30936.507,E2 30936.507} C_VEL
LIN {X 0,Y 651.993,Z 345.891,A -85,B 0,C 180,E1 30936.392,E2 30936.392} C_VEL
LIN {X 0,Y 649.594,Z 343.116,A -85,B 0,C 180,E1 30936.107,E2 30936.107} C_VEL
LIN {X 0,Y 648.819,Z 340.938,A -85,B 0,C 180,E1 30935.92,E2 30935.92} C_VEL
LIN {X 0,Y 648.72,Z 340.426,A -85,B 0,C 180,E1 30935.631,E2 30935.631} C_VEL
LIN {X 0,Y 648.764,Z 340.42,A -85,B 0,C 180,E1 30932.659,E2 30932.659} C_VEL
LIN {X 0,Y 648.733,Z 340.423,A -85,B 0,C 180,E1 30929.53,E2 30929.53} C_VEL
LIN {X 0,Y 648.769,Z 340.421,A -85,B 0,C 180,E1 30926.489,E2 30926.489} C_VEL
LIN {X 0,Y 648.796,Z 340.658,A -85,B 0,C 180,E1 30924.291,E2 30924.291} C_VEL
LIN {X 0,Y 650.089,Z 343.935,A -85,B 0,C 180,E1 30923.908,E2 30923.908} C_VEL
LIN {X 0,Y 655.649,Z 356.651,A -85,B 0,C 180,E1 30922.629,E2 30922.629} C_VEL
LIN {X 0,Y 662.86,Z 373.639,A -85,B 0,C 180,E1 30921.133,E2 30921.133} C_VEL
LIN {X 0,Y 671.148,Z 387.447,A -85,B 0,C 180,E1 30919.883,E2 30919.883} C_VEL
LIN {X 0,Y 672.107,Z 427.382,A -85,B 0,C 180,E1 30917.73,E2 30917.73} C_VEL
LIN {X 0,Y 678.023,Z 453.928,A -85,B 0,C 180,E1 30916.829,E2 30916.829} C_VEL
LIN {X 0,Y 678.285,Z 457.049,A -85,B 0,C 180,E1 30916.758,E2 30916.758} C_VEL
LIN {X 0,Y 674.972,Z 661.216,A -85,B 0,C 180,E1 30914.02,E2 30914.02} C_VEL
LIN {X 0,Y 671.589,Z 885.871,A -85,B 0,C 180,E1 30911.097,E2 30911.097} C_VEL
LIN {X 0,Y 670.763,Z 917.556,A -85,B 0,C 180,E1 30910.627,E2 30910.627} C_VEL
LIN {X 0,Y 669.778,Z 941.601,A -85,B 0,C 180,E1 30910.127,E2 30910.127} C_VEL
LIN {X 0,Y 668.608,Z 965.417,A -85,B 0,C 180,E1 30909.498,E2 30909.498} C_VEL
LIN {X 0,Y 666.965,Z 993.163,A -85,B 0,C 180,E1 30908.583,E2 30908.583} C_VEL
LIN {X 0,Y 665.416,Z 1016.126,A -85,B 0,C 180,E1 30907.665,E2 30907.665} C_VEL
LIN {X 0,Y 663.855,Z 1037.708,A -85,B 0,C 180,E1 30906.669,E2 30906.669} C_VEL
LIN {X 0,Y 662.097,Z 1060.897,A -85,B 0,C 180,E1 30905.444,E2 30905.444} C_VEL
LIN {X 0,Y 660.055,Z 1085.596,A -85,B 0,C 180,E1 30903.933,E2 30903.933} C_VEL
LIN {X 0,Y 658.45,Z 1104.573,A -85,B 0,C 180,E1 30902.621,E2 30902.621} C_VEL
LIN {X 0,Y 656.871,Z 1123.474,A -85,B 0,C 180,E1 30901.167,E2 30901.167} C_VEL
LIN {X 0,Y 655.017,Z 1146.44,A -85,B 0,C 180,E1 30899.171,E2 30899.171} C_VEL
LIN {X 0,Y 653.648,Z 1163.385,A -85,B 0,C 180,E1 30897.514,E2 30897.514} C_VEL
LIN {X 0,Y 652.377,Z 1180.074,A -85,B 0,C 180,E1 30895.705,E2 30895.705} C_VEL
LIN {X 0,Y 651.149,Z 1197.853,A -85,B 0,C 180,E1 30893.531,E2 30893.531} C_VEL
LIN {X 0,Y 650.302,Z 1211.468,A -85,B 0,C 180,E1 30891.655,E2 30891.655} C_VEL
LIN {X 0,Y 649.598,Z 1224.162,A -85,B 0,C 180,E1 30889.7,E2 30889.7} C_VEL
LIN {X 0,Y 648.949,Z 1237.817,A -85,B 0,C 180,E1 30887.299,E2 30887.299} C_VEL
LIN {X 0,Y 648.525,Z 1248.199,A -85,B 0,C 180,E1 30885.167,E2 30885.167} C_VEL
LIN {X 0,Y 648.264,Z 1256.515,A -85,B 0,C 180,E1 30883.195,E2 30883.195} C_VEL
LIN {X 0,Y 648.09,Z 1263.662,A -85,B 0,C 180,E1 30881.209,E2 30881.209} C_VEL
LIN {X 0,Y 647.974,Z 1270.816,A -85,B 0,C 180,E1 30878.787,E2 30878.787} C_VEL
LIN {X 0,Y 647.939,Z 1276.096,A -85,B 0,C 180,E1 30876.375,E2 30876.375} C_VEL
LIN {X 0,Y 647.919,Z 1279.476,A -85,B 0,C 180,E1 30874.159,E2 30874.159} C_VEL
LIN {X 0,Y 647.909,Z 1281.601,A -85,B 0,C 180,E1 30871.592,E2 30871.592} C_VEL
LIN {X 0,Y 647.867,Z 1281.872,A -85,B 0,C 180,E1 30869.469,E2 30869.469} C_VEL
LIN {X 0,Y 647.907,Z 1281.014,A -85,B 0,C 180,E1 30867.523,E2 30867.523} C_VEL
LIN {X 0,Y 647.913,Z 1279.021,A -85,B 0,C 180,E1 30865.486,E2 30865.486} C_VEL
LIN {X 0,Y 647.936,Z 1275.25,A -85,B 0,C 180,E1 30863.176,E2 30863.176} C_VEL
LIN {X 0,Y 647.956,Z 1269.838,A -85,B 0,C 180,E1 30860.855,E2 30860.855} C_VEL
LIN {X 0,Y 648.1,Z 1263.357,A -85,B 0,C 180,E1 30858.701,E2 30858.701} C_VEL
LIN {X 0,Y 648.263,Z 1256.513,A -85,B 0,C 180,E1 30856.805,E2 30856.805} C_VEL
LIN {X 0,Y 648.528,Z 1248.076,A -85,B 0,C 180,E1 30854.805,E2 30854.805} C_VEL
LIN {X 0,Y 648.97,Z 1237.353,A -85,B 0,C 180,E1 30852.609,E2 30852.609} C_VEL
LIN {X 0,Y 649.599,Z 1224.163,A -85,B 0,C 180,E1 30850.3,E2 30850.3} C_VEL
LIN {X 0,Y 650.302,Z 1211.467,A -85,B 0,C 180,E1 30848.345,E2 30848.345} C_VEL
LIN {X 0,Y 651.204,Z 1197.14,A -85,B 0,C 180,E1 30846.375,E2 30846.375} C_VEL
LIN {X 0,Y 652.431,Z 1179.228,A -85,B 0,C 180,E1 30844.199,E2 30844.199} C_VEL
LIN {X 0,Y 653.683,Z 1162.992,A -85,B 0,C 180,E1 30842.446,E2 30842.446} C_VEL
LIN {X 0,Y 655.122,Z 1145.228,A -85,B 0,C 180,E1 30840.715,E2 30840.715} C_VEL
LIN {X 0,Y 656.895,Z 1123.184,A -85,B 0,C 180,E1 30838.809,E2 30838.809} C_VEL
LIN {X 0,Y 658.45,Z 1104.569,A -85,B 0,C 180,E1 30837.379,E2 30837.379} C_VEL
LIN {X 0,Y 660.122,Z 1084.854,A -85,B 0,C 180,E1 30836.019,E2 30836.019} C_VEL
LIN {X 0,Y 662.159,Z 1060.004,A -85,B 0,C 180,E1 30834.507,E2 30834.507} C_VEL
LIN {X 0,Y 663.857,Z 1037.712,A -85,B 0,C 180,E1 30833.331,E2 30833.331} C_VEL
LIN {X 0,Y 665.417,Z 1016.126,A -85,B 0,C 180,E1 30832.335,E2 30832.335} C_VEL
LIN {X 0,Y 667.108,Z 991.198,A -85,B 0,C 180,E1 30831.343,E2 30831.343} C_VEL
LIN {X 0,Y 668.679,Z 963.989,A -85,B 0,C 180,E1 30830.461,E2 30830.461} C_VEL
LIN {X 0,Y 669.814,Z 940.82,A -85,B 0,C 180,E1 30829.854,E2 30829.854} C_VEL
LIN {X 0,Y 670.849,Z 915.411,A -85,B 0,C 180,E1 30829.333,E2 30829.333} C_VEL
LIN {X 0,Y 671.67,Z 880.368,A -85,B 0,C 180,E1 30828.833,E2 30828.833} C_VEL
LIN {X 0,Y 675.059,Z 655.736,A -85,B 0,C 180,E1 30825.908,E2 30825.908} C_VEL
LIN {X 0,Y 678.304,Z 455.217,A -85,B 0,C 180,E1 30823.216,E2 30823.216} C_VEL
LIN {X 0,Y 672.151,Z 426.246,A -85,B 0,C 180,E1 30822.199,E2 30822.199} C_VEL
LIN {X 0,Y 673.673,Z 389.19,A -85,B 0,C 180,E1 30819.826,E2 30819.826} C_VEL
LIN {X 0,Y 659.903,Z 362.263,A -85,B 0,C 180,E1 30816.547,E2 30816.547} C_VEL
LIN {X 0,Y 653.15,Z 349.338,A -85,B 0,C 180,E1 30814.821,E2 30814.821} C_VEL
LIN {X 0,Y 650.468,Z 344.44,A -85,B 0,C 180,E1 30814.13,E2 30814.13} C_VEL
LIN {X 0,Y 648.816,Z 340.819,A -85,B 0,C 180,E1 30813.624,E2 30813.624} C_VEL
LIN {X 0,Y 648.755,Z 340.412,A -85,B 0,C 180,E1 30812.961,E2 30812.961} C_VEL
LIN {X 0,Y 648.765,Z 340.42,A -85,B 0,C 180,E1 30809.808,E2 30809.808} C_VEL
LIN {X 0,Y 648.752,Z 340.412,A -85,B 0,C 180,E1 30806.747,E2 30806.747} C_VEL
LIN {X 0,Y 648.764,Z 340.407,A -85,B 0,C 180,E1 30803.623,E2 30803.623} C_VEL
LIN {X 0,Y 648.751,Z 340.414,A -85,B 0,C 180,E1 30800.573,E2 30800.573} C_VEL
LIN {X 0,Y 648.765,Z 340.409,A -85,B 0,C 180,E1 30797.446,E2 30797.446} C_VEL
LIN {X 0,Y 648.746,Z 340.418,A -85,B 0,C 180,E1 30794.368,E2 30794.368} C_VEL
LIN {X 0,Y 648.766,Z 340.407,A -85,B 0,C 180,E1 30791.288,E2 30791.288} C_VEL
LIN {X 0,Y 648.741,Z 340.416,A -85,B 0,C 180,E1 30788.152,E2 30788.152} C_VEL
LIN {X 0,Y 648.767,Z 340.405,A -85,B 0,C 180,E1 30785.129,E2 30785.129} C_VEL
LIN {X 0,Y 648.742,Z 340.411,A -85,B 0,C 180,E1 30782.032,E2 30782.032} C_VEL
LIN {X 0,Y 648.769,Z 340.413,A -85,B 0,C 180,E1 30778.94,E2 30778.94} C_VEL
LIN {X 0,Y 648.736,Z 340.418,A -85,B 0,C 180,E1 30775.757,E2 30775.757} C_VEL
LIN {X 0,Y 648.772,Z 340.411,A -85,B 0,C 180,E1 30772.74,E2 30772.74} C_VEL
LIN {X 0,Y 648.736,Z 340.42,A -85,B 0,C 180,E1 30769.611,E2 30769.611} C_VEL
LIN {X 0,Y 648.768,Z 340.413,A -85,B 0,C 180,E1 30766.542,E2 30766.542} C_VEL
LIN {X 0,Y 648.731,Z 340.415,A -85,B 0,C 180,E1 30763.433,E2 30763.433} C_VEL
LIN {X 0,Y 648.757,Z 340.414,A -85,B 0,C 180,E1 30760.461,E2 30760.461} C_VEL
LIN {X 0,Y 648.736,Z 340.415,A -85,B 0,C 180,E1 30757.336,E2 30757.336} C_VEL
LIN {X 0,Y 648.745,Z 340.415,A -85,B 0,C 180,E1 30754.373,E2 30754.373} C_VEL
LIN {X 0,Y 648.734,Z 340.416,A -85,B 0,C 180,E1 30751.156,E2 30751.156} C_VEL
LIN {X 0,Y 648.731,Z 340.416,A -85,B 0,C 180,E1 30748.292,E2 30748.292} C_VEL
LIN {X 0,Y 648.74,Z 340.418,A -85,B 0,C 180,E1 30745.08,E2 30745.08} C_VEL
LIN {X 0,Y 648.724,Z 340.417,A -85,B 0,C 180,E1 30742.161,E2 30742.161} C_VEL
LIN {X 0,Y 648.745,Z 340.419,A -85,B 0,C 180,E1 30738.96,E2 30738.96} C_VEL
LIN {X 0,Y 648.77,Z 340.411,A -85,B 0,C 180,E1 30737.475,E2 30737.475} C_VEL
LIN {X 0,Y 647.799,Z 340.539,A -85,B 0,C 180,E1 30736.795,E2 30736.795} C_VEL
LIN {X 0,Y 641.319,Z 341.344,A -85,B 0,C 180,E1 30734.888,E2 30734.888} C_VEL
LIN {X 0,Y 640.774,Z 341.408,A -85,B 0,C 180,E1 30734.392,E2 30734.392} C_VEL
LIN {X 0,Y 640.823,Z 341.4,A -85,B 0,C 180,E1 30731.419,E2 30731.419} C_VEL
LIN {X 0,Y 640.779,Z 341.408,A -85,B 0,C 180,E1 30728.392,E2 30728.392} C_VEL
LIN {X 0,Y 640.781,Z 341.404,A -85,B 0,C 180,E1 30725.593,E2 30725.593} C_VEL
LIN {X 0,Y 640.786,Z 341.407,A -85,B 0,C 180,E1 30722.358,E2 30722.358} C_VEL
LIN {X 0,Y 640.764,Z 341.404,A -85,B 0,C 180,E1 30719.636,E2 30719.636} C_VEL
LIN {X 0,Y 640.83,Z 341.402,A -85,B 0,C 180,E1 30716.603,E2 30716.603} C_VEL
LIN {X 0,Y 640.758,Z 341.402,A -85,B 0,C 180,E1 30713.643,E2 30713.643} C_VEL
LIN {X 0,Y 640.819,Z 341.403,A -85,B 0,C 180,E1 30710.744,E2 30710.744} C_VEL
LIN {X 0,Y 640.763,Z 341.41,A -85,B 0,C 180,E1 30707.715,E2 30707.715} C_VEL
LIN {X 0,Y 640.766,Z 341.405,A -85,B 0,C 180,E1 30704.999,E2 30704.999} C_VEL
LIN {X 0,Y 640.78,Z 341.414,A -85,B 0,C 180,E1 30701.795,E2 30701.795} C_VEL
LIN {X 0,Y 640.749,Z 341.412,A -85,B 0,C 180,E1 30699.068,E2 30699.068} C_VEL
LIN {X 0,Y 640.834,Z 341.409,A -85,B 0,C 180,E1 30696.09,E2 30696.09} C_VEL
LIN {X 0,Y 640.747,Z 341.41,A -85,B 0,C 180,E1 30693.131,E2 30693.131} C_VEL
LIN {X 0,Y 640.765,Z 341.41,A -85,B 0,C 180,E1 30690.447,E2 30690.447} C_VEL
LIN {X 0,Y 640.757,Z 341.39,A -85,B 0,C 180,E1 30687.227,E2 30687.227} C_VEL
LIN {X 0,Y 640.744,Z 341.415,A -85,B 0,C 180,E1 30684.538,E2 30684.538} C_VEL
LIN {X 0,Y 640.821,Z 341.402,A -85,B 0,C 180,E1 30681.566,E2 30681.566} C_VEL
LIN {X 0,Y 640.735,Z 341.397,A -85,B 0,C 180,E1 30678.66,E2 30678.66} C_VEL
LIN {X 0,Y 640.744,Z 341.361,A -85,B 0,C 180,E1 30676.083,E2 30676.083} C_VEL
LIN {X 0,Y 640.79,Z 341.615,A -85,B 0,C 180,E1 30674.942,E2 30674.942} C_VEL
LIN {X 0,Y 641.179,Z 343.145,A -85,B 0,C 180,E1 30674.754,E2 30674.754} C_VEL
LIN {X 0,Y 643.159,Z 346.155,A -85,B 0,C 180,E1 30674.491,E2 30674.491} C_VEL
LIN {X 0,Y 644.895,Z 347.876,A -85,B 0,C 180,E1 30674.28,E2 30674.28} C_VEL
LIN {X 0,Y 647.445,Z 351.635,A -85,B 0,C 180,E1 30673.952,E2 30673.952} C_VEL
LIN {X 0,Y 649.08,Z 353.589,A -85,B 0,C 180,E1 30673.753,E2 30673.753} C_VEL
LIN {X 0,Y 663.936,Z 373.843,A -85,B 0,C 180,E1 30671.995,E2 30671.995} C_VEL
LIN {X 0,Y 671.43,Z 384.592,A -85,B 0,C 180,E1 30671.152,E2 30671.152} C_VEL
LIN {X 0,Y 667.694,Z 602.467,A -85,B 0,C 180,E1 30668.246,E2 30668.246} C_VEL
LIN {X 0,Y 665.075,Z 757.405,A -85,B 0,C 180,E1 30666.207,E2 30666.207} C_VEL
LIN {X 0,Y 664.02,Z 783.588,A -85,B 0,C 180,E1 30665.717,E2 30665.717} C_VEL
LIN {X 0,Y 662.626,Z 810.737,A -85,B 0,C 180,E1 30665.036,E2 30665.036} C_VEL
LIN {X 0,Y 661.04,Z 837.082,A -85,B 0,C 180,E1 30664.199,E2 30664.199} C_VEL
LIN {X 0,Y 659.158,Z 863.617,A -85,B 0,C 180,E1 30663.17,E2 30663.17} C_VEL
LIN {X 0,Y 657.275,Z 887.649,A -85,B 0,C 180,E1 30662.06,E2 30662.06} C_VEL
LIN {X 0,Y 655.285,Z 911.699,A -85,B 0,C 180,E1 30660.773,E2 30660.773} C_VEL
LIN {X 0,Y 653.193,Z 935.466,A -85,B 0,C 180,E1 30659.308,E2 30659.308} C_VEL
LIN {X 0,Y 651.229,Z 956.848,A -85,B 0,C 180,E1 30657.807,E2 30657.807} C_VEL
LIN {X 0,Y 649.207,Z 979.465,A -85,B 0,C 180,E1 30656.008,E2 30656.008} C_VEL
LIN {X 0,Y 647.291,Z 1001.026,A -85,B 0,C 180,E1 30654.056,E2 30654.056} C_VEL
LIN {X 0,Y 645.59,Z 1020.796,A -85,B 0,C 180,E1 30652.031,E2 30652.031} C_VEL
LIN {X 0,Y 644.206,Z 1038.177,A -85,B 0,C 180,E1 30650.016,E2 30650.016} C_VEL
LIN {X 0,Y 643.024,Z 1054.565,A -85,B 0,C 180,E1 30647.879,E2 30647.879} C_VEL
LIN {X 0,Y 642.019,Z 1070.057,A -85,B 0,C 180,E1 30645.57,E2 30645.57} C_VEL
LIN {X 0,Y 641.335,Z 1082.11,A -85,B 0,C 180,E1 30643.535,E2 30643.535} C_VEL
LIN {X 0,Y 640.77,Z 1093.666,A -85,B 0,C 180,E1 30641.306,E2 30641.306} C_VEL
LIN {X 0,Y 640.373,Z 1104.569,A -85,B 0,C 180,E1 30638.819,E2 30638.819} C_VEL
LIN {X 0,Y 640.144,Z 1112.603,A -85,B 0,C 180,E1 30636.632,E2 30636.632} C_VEL
LIN {X 0,Y 640.014,Z 1119.538,A -85,B 0,C 180,E1 30634.332,E2 30634.332} C_VEL
LIN {X 0,Y 639.941,Z 1125.065,A -85,B 0,C 180,E1 30631.961,E2 30631.961} C_VEL
LIN {X 0,Y 639.913,Z 1128.955,A -85,B 0,C 180,E1 30629.588,E2 30629.588} C_VEL
LIN {X 0,Y 639.871,Z 1131.138,A -85,B 0,C 180,E1 30627.35,E2 30627.35} C_VEL
LIN {X 0,Y 639.907,Z 1132,A -85,B 0,C 180,E1 30624.954,E2 30624.954} C_VEL
LIN {X 0,Y 639.872,Z 1131.136,A -85,B 0,C 180,E1 30622.556,E2 30622.556} C_VEL
LIN {X 0,Y 639.913,Z 1128.918,A -85,B 0,C 180,E1 30620.297,E2 30620.297} C_VEL
LIN {X 0,Y 639.945,Z 1125.002,A -85,B 0,C 180,E1 30617.913,E2 30617.913} C_VEL
LIN {X 0,Y 640.017,Z 1119.322,A -85,B 0,C 180,E1 30615.495,E2 30615.495} C_VEL
LIN {X 0,Y 640.164,Z 1112.277,A -85,B 0,C 180,E1 30613.182,E2 30613.182} C_VEL
LIN {X 0,Y 640.396,Z 1104.145,A -85,B 0,C 180,E1 30610.981,E2 30610.981} C_VEL
LIN {X 0,Y 640.823,Z 1092.767,A -85,B 0,C 180,E1 30608.417,E2 30608.417} C_VEL
LIN {X 0,Y 641.365,Z 1081.476,A -85,B 0,C 180,E1 30606.265,E2 30606.265} C_VEL
LIN {X 0,Y 642.117,Z 1068.645,A -85,B 0,C 180,E1 30604.108,E2 30604.108} C_VEL
LIN {X 0,Y 643.15,Z 1052.768,A -85,B 0,C 180,E1 30601.782,E2 30601.782} C_VEL
LIN {X 0,Y 644.313,Z 1036.837,A -85,B 0,C 180,E1 30599.733,E2 30599.733} C_VEL
LIN {X 0,Y 645.791,Z 1018.258,A -85,B 0,C 180,E1 30597.604,E2 30597.604} C_VEL
LIN {X 0,Y 647.467,Z 999.014,A -85,B 0,C 180,E1 30595.66,E2 30595.66} C_VEL
LIN {X 0,Y 649.353,Z 977.939,A -85,B 0,C 180,E1 30593.768,E2 30593.768} C_VEL
LIN {X 0,Y 651.349,Z 955.665,A -85,B 0,C 180,E1 30592.014,E2 30592.014} C_VEL
LIN {X 0,Y 653.411,Z 933.03,A -85,B 0,C 180,E1 30590.443,E2 30590.443} C_VEL
LIN {X 0,Y 655.518,Z 908.637,A -85,B 0,C 180,E1 30588.964,E2 30588.964} C_VEL
LIN {X 0,Y 657.436,Z 885.676,A -85,B 0,C 180,E1 30587.751,E2 30587.751} C_VEL
LIN {X 0,Y 659.368,Z 860.895,A -85,B 0,C 180,E1 30586.629,E2 30586.629} C_VEL
LIN {X 0,Y 661.149,Z 834.972,A -85,B 0,C 180,E1 30585.639,E2 30585.639} C_VEL
LIN {X 0,Y 662.633,Z 810.757,A -85,B 0,C 180,E1 30584.873,E2 30584.873} C_VEL
LIN {X 0,Y 664.004,Z 783.74,A -85,B 0,C 180,E1 30584.198,E2 30584.198} C_VEL
LIN {X 0,Y 665.057,Z 757.899,A -85,B 0,C 180,E1 30583.71,E2 30583.71} C_VEL
LIN {X 0,Y 666.851,Z 654.496,A -85,B 0,C 180,E1 30582.347,E2 30582.347} C_VEL
LIN {X 0,Y 670.561,Z 433.567,A -85,B 0,C 180,E1 30579.419,E2 30579.419} C_VEL
LIN {X 0,Y 671.277,Z 384.157,A -85,B 0,C 180,E1 30578.738,E2 30578.738} C_VEL
LIN {X 0,Y 658.758,Z 366.968,A -85,B 0,C 180,E1 30577.372,E2 30577.372} C_VEL
LIN {X 0,Y 648.644,Z 353.014,A -85,B 0,C 180,E1 30576.187,E2 30576.187} C_VEL
LIN {X 0,Y 645.299,Z 348.646,A -85,B 0,C 180,E1 30575.764,E2 30575.764} C_VEL
LIN {X 0,Y 644.332,Z 347.116,A -85,B 0,C 180,E1 30575.631,E2 30575.631} C_VEL
LIN {X 0,Y 641.834,Z 344.502,A -85,B 0,C 180,E1 30575.309,E2 30575.309} C_VEL
LIN {X 0,Y 640.885,Z 341.996,A -85,B 0,C 180,E1 30575.087,E2 30575.087} C_VEL
LIN {X 0,Y 640.816,Z 341.417,A -85,B 0,C 180,E1 30574.821,E2 30574.821} C_VEL
LIN {X 0,Y 640.795,Z 341.413,A -85,B 0,C 180,E1 30571.648,E2 30571.648} C_VEL
LIN {X 0,Y 640.827,Z 341.41,A -85,B 0,C 180,E1 30568.695,E2 30568.695} C_VEL
LIN {X 0,Y 640.804,Z 341.413,A -85,B 0,C 180,E1 30565.473,E2 30565.473} C_VEL
LIN {X 0,Y 640.874,Z 341.846,A -85,B 0,C 180,E1 30564.91,E2 30564.91} C_VEL
LIN {X 0,Y 642.266,Z 345.097,A -85,B 0,C 180,E1 30564.501,E2 30564.501} C_VEL
LIN {X 0,Y 646.529,Z 354.551,A -85,B 0,C 180,E1 30563.457,E2 30563.457} C_VEL
LIN {X 0,Y 652.145,Z 368.277,A -85,B 0,C 180,E1 30562.148,E2 30562.148} C_VEL
LIN {X 0,Y 657.023,Z 379.192,A -85,B 0,C 180,E1 30561.171,E2 30561.171} C_VEL
LIN {X 0,Y 664.152,Z 390.941,A -85,B 0,C 180,E1 30560.079,E2 30560.079} C_VEL
LIN {X 0,Y 664.79,Z 422.682,A -85,B 0,C 180,E1 30558.348,E2 30558.348} C_VEL
LIN {X 0,Y 668.945,Z 441.306,A -85,B 0,C 180,E1 30557.773,E2 30557.773} C_VEL
LIN {X 0,Y 672.779,Z 458.18,A -85,B 0,C 180,E1 30557.242,E2 30557.242} C_VEL
LIN {X 0,Y 669.198,Z 662.286,A -85,B 0,C 180,E1 30554.484,E2 30554.484} C_VEL
LIN {X 0,Y 665.543,Z 886.863,A -85,B 0,C 180,E1 30551.538,E2 30551.538} C_VEL
LIN {X 0,Y 664.665,Z 917.725,A -85,B 0,C 180,E1 30551.076,E2 30551.076} C_VEL
LIN {X 0,Y 663.625,Z 941.489,A -85,B 0,C 180,E1 30550.579,E2 30550.579} C_VEL
LIN {X 0,Y 662.402,Z 964.687,A -85,B 0,C 180,E1 30549.965,E2 30549.965} C_VEL
LIN {X 0,Y 660.702,Z 991.923,A -85,B 0,C 180,E1 30549.071,E2 30549.071} C_VEL
LIN {X 0,Y 658.992,Z 1015.334,A -85,B 0,C 180,E1 30548.136,E2 30548.136} C_VEL
LIN {X 0,Y 657.324,Z 1036.732,A -85,B 0,C 180,E1 30547.147,E2 30547.147} C_VEL
LIN {X 0,Y 655.547,Z 1058.229,A -85,B 0,C 180,E1 30546.014,E2 30546.014} C_VEL
LIN {X 0,Y 653.371,Z 1083.39,A -85,B 0,C 180,E1 30544.487,E2 30544.487} C_VEL
LIN {X 0,Y 651.51,Z 1103.784,A -85,B 0,C 180,E1 30543.074,E2 30543.074} C_VEL
LIN {X 0,Y 649.827,Z 1122.265,A -85,B 0,C 180,E1 30541.647,E2 30541.647} C_VEL
LIN {X 0,Y 648.008,Z 1142.953,A -85,B 0,C 180,E1 30539.867,E2 30539.867} C_VEL
LIN {X 0,Y 646.298,Z 1162.457,A -85,B 0,C 180,E1 30537.954,E2 30537.954} C_VEL
LIN {X 0,Y 644.956,Z 1178.382,A -85,B 0,C 180,E1 30536.221,E2 30536.221} C_VEL
LIN {X 0,Y 643.598,Z 1196.541,A -85,B 0,C 180,E1 30534.004,E2 30534.004} C_VEL
LIN {X 0,Y 642.554,Z 1211.47,A -85,B 0,C 180,E1 30531.929,E2 30531.929} C_VEL
LIN {X 0,Y 641.769,Z 1224.16,A -85,B 0,C 180,E1 30529.95,E2 30529.95} C_VEL
LIN {X 0,Y 641.052,Z 1237.819,A -85,B 0,C 180,E1 30527.519,E2 30527.519} C_VEL
LIN {X 0,Y 640.591,Z 1248.078,A -85,B 0,C 180,E1 30525.388,E2 30525.388} C_VEL
LIN {X 0,Y 640.295,Z 1256.158,A -85,B 0,C 180,E1 30523.455,E2 30523.455} C_VEL
LIN {X 0,Y 640.137,Z 1263.056,A -85,B 0,C 180,E1 30521.533,E2 30521.533} C_VEL
LIN {X 0,Y 639.969,Z 1269.33,A -85,B 0,C 180,E1 30519.442,E2 30519.442} C_VEL
LIN {X 0,Y 639.95,Z 1274.739,A -85,B 0,C 180,E1 30517.179,E2 30517.179} C_VEL
LIN {X 0,Y 639.914,Z 1278.792,A -85,B 0,C 180,E1 30514.75,E2 30514.75} C_VEL
LIN {X 0,Y 639.908,Z 1280.879,A -85,B 0,C 180,E1 30512.687,E2 30512.687} C_VEL
LIN {X 0,Y 639.868,Z 1281.782,A -85,B 0,C 180,E1 30510.895,E2 30510.895} C_VEL
LIN {X 0,Y 639.868,Z 1281.782,A -85,B 0,C 180,E1 30509.105,E2 30509.105} C_VEL
LIN {X 0,Y 639.908,Z 1280.879,A -85,B 0,C 180,E1 30507.313,E2 30507.313} C_VEL
LIN {X 0,Y 639.914,Z 1278.791,A -85,B 0,C 180,E1 30505.25,E2 30505.25} C_VEL
LIN {X 0,Y 639.951,Z 1274.734,A -85,B 0,C 180,E1 30502.82,E2 30502.82} C_VEL
LIN {X 0,Y 639.969,Z 1269.329,A -85,B 0,C 180,E1 30500.558,E2 30500.558} C_VEL
LIN {X 0,Y 640.137,Z 1263.054,A -85,B 0,C 180,E1 30498.467,E2 30498.467} C_VEL
LIN {X 0,Y 640.294,Z 1256.156,A -85,B 0,C 180,E1 30496.545,E2 30496.545} C_VEL
LIN {X 0,Y 640.591,Z 1248.077,A -85,B 0,C 180,E1 30494.612,E2 30494.612} C_VEL
LIN {X 0,Y 641.092,Z 1236.89,A -85,B 0,C 180,E1 30492.294,E2 30492.294} C_VEL
LIN {X 0,Y 641.8,Z 1223.588,A -85,B 0,C 180,E1 30489.956,E2 30489.956} C_VEL
LIN {X 0,Y 642.598,Z 1210.824,A -85,B 0,C 180,E1 30487.976,E2 30487.976} C_VEL
LIN {X 0,Y 643.747,Z 1194.676,A -85,B 0,C 180,E1 30485.749,E2 30485.749} C_VEL
LIN {X 0,Y 645.03,Z 1177.535,A -85,B 0,C 180,E1 30483.683,E2 30483.683} C_VEL
LIN {X 0,Y 646.373,Z 1161.524,A -85,B 0,C 180,E1 30481.949,E2 30481.949} C_VEL
LIN {X 0,Y 648.112,Z 1141.591,A -85,B 0,C 180,E1 30480.01,E2 30480.01} C_VEL
LIN {X 0,Y 649.886,Z 1121.636,A -85,B 0,C 180,E1 30478.302,E2 30478.302} C_VEL
LIN {X 0,Y 651.562,Z 1103.23,A -85,B 0,C 180,E1 30476.886,E2 30476.886} C_VEL
LIN {X 0,Y 653.534,Z 1081.68,A -85,B 0,C 180,E1 30475.399,E2 30475.399} C_VEL
LIN {X 0,Y 655.623,Z 1057.243,A -85,B 0,C 180,E1 30473.931,E2 30473.931} C_VEL
LIN {X 0,Y 657.327,Z 1036.703,A -85,B 0,C 180,E1 30472.851,E2 30472.851} C_VEL
LIN {X 0,Y 659.054,Z 1014.55,A -85,B 0,C 180,E1 30471.83,E2 30471.83} C_VEL
LIN {X 0,Y 661.017,Z 987.13,A -85,B 0,C 180,E1 30470.758,E2 30470.758} C_VEL
LIN {X 0,Y 662.51,Z 962.582,A -85,B 0,C 180,E1 30469.974,E2 30469.974} C_VEL
LIN {X 0,Y 663.707,Z 939.757,A -85,B 0,C 180,E1 30469.38,E2 30469.38} C_VEL
LIN {X 0,Y 664.85,Z 913.393,A -85,B 0,C 180,E1 30468.845,E2 30468.845} C_VEL
LIN {X 0,Y 665.731,Z 875.024,A -85,B 0,C 180,E1 30468.309,E2 30468.309} C_VEL
LIN {X 0,Y 669.415,Z 649.81,A -85,B 0,C 180,E1 30465.351,E2 30465.351} C_VEL
LIN {X 0,Y 672.773,Z 457.261,A -85,B 0,C 180,E1 30462.744,E2 30462.744} C_VEL
LIN {X 0,Y 666.003,Z 425.234,A -85,B 0,C 180,E1 30461.613,E2 30461.613} C_VEL
LIN {X 0,Y 667.374,Z 393.487,A -85,B 0,C 180,E1 30459.55,E2 30459.55} C_VEL
LIN {X 0,Y 654.289,Z 367.607,A -85,B 0,C 180,E1 30456.367,E2 30456.367} C_VEL
LIN {X 0,Y 647.553,Z 354.754,A -85,B 0,C 180,E1 30454.627,E2 30454.627} C_VEL
LIN {X 0,Y 644.893,Z 349.863,A -85,B 0,C 180,E1 30453.93,E2 30453.93} C_VEL
LIN {X 0,Y 642.642,Z 345.564,A -85,B 0,C 180,E1 30453.315,E2 30453.315} C_VEL
LIN {X 0,Y 641.06,Z 342.619,A -85,B 0,C 180,E1 30452.874,E2 30452.874} C_VEL
LIN {X 0,Y 640.826,Z 341.544,A -85,B 0,C 180,E1 30452.675,E2 30452.675} C_VEL
LIN {X 0,Y 640.82,Z 341.407,A -85,B 0,C 180,E1 30449.645,E2 30449.645} C_VEL
LIN {X 0,Y 640.808,Z 341.4,A -85,B 0,C 180,E1 30446.604,E2 30446.604} C_VEL
LIN {X 0,Y 640.823,Z 341.396,A -85,B 0,C 180,E1 30443.543,E2 30443.543} C_VEL
LIN {X 0,Y 640.805,Z 341.404,A -85,B 0,C 180,E1 30440.458,E2 30440.458} C_VEL
LIN {X 0,Y 640.827,Z 341.398,A -85,B 0,C 180,E1 30437.432,E2 30437.432} C_VEL
LIN {X 0,Y 640.804,Z 341.408,A -85,B 0,C 180,E1 30434.273,E2 30434.273} C_VEL
LIN {X 0,Y 640.827,Z 341.396,A -85,B 0,C 180,E1 30431.247,E2 30431.247} C_VEL
LIN {X 0,Y 640.803,Z 341.404,A -85,B 0,C 180,E1 30428.163,E2 30428.163} C_VEL
LIN {X 0,Y 640.828,Z 341.394,A -85,B 0,C 180,E1 30425.103,E2 30425.103} C_VEL
LIN {X 0,Y 640.8,Z 341.399,A -85,B 0,C 180,E1 30421.967,E2 30421.967} C_VEL
LIN {X 0,Y 640.831,Z 341.402,A -85,B 0,C 180,E1 30418.927,E2 30418.927} C_VEL
LIN {X 0,Y 640.799,Z 341.408,A -85,B 0,C 180,E1 30415.794,E2 30415.794} C_VEL
LIN {X 0,Y 640.834,Z 341.4,A -85,B 0,C 180,E1 30412.739,E2 30412.739} C_VEL
LIN {X 0,Y 640.795,Z 341.408,A -85,B 0,C 180,E1 30409.572,E2 30409.572} C_VEL
LIN {X 0,Y 640.828,Z 341.402,A -85,B 0,C 180,E1 30406.556,E2 30406.556} C_VEL
LIN {X 0,Y 640.791,Z 341.403,A -85,B 0,C 180,E1 30403.408,E2 30403.408} C_VEL
LIN {X 0,Y 640.823,Z 341.403,A -85,B 0,C 180,E1 30400.399,E2 30400.399} C_VEL
LIN {X 0,Y 640.79,Z 341.403,A -85,B 0,C 180,E1 30397.233,E2 30397.233} C_VEL
LIN {X 0,Y 640.812,Z 341.404,A -85,B 0,C 180,E1 30394.292,E2 30394.292} C_VEL
LIN {X 0,Y 640.789,Z 341.404,A -85,B 0,C 180,E1 30391.071,E2 30391.071} C_VEL
LIN {X 0,Y 640.804,Z 341.405,A -85,B 0,C 180,E1 30388.17,E2 30388.17} C_VEL
LIN {X 0,Y 640.79,Z 341.406,A -85,B 0,C 180,E1 30384.954,E2 30384.954} C_VEL
LIN {X 0,Y 640.792,Z 341.406,A -85,B 0,C 180,E1 30382.063,E2 30382.063} C_VEL
LIN {X 0,Y 640.788,Z 341.406,A -85,B 0,C 180,E1 30378.773,E2 30378.773} C_VEL
LIN {X 0,Y 640.79,Z 341.406,A -85,B 0,C 180,E1 30375.871,E2 30375.871} C_VEL
LIN {X 0,Y 640.774,Z 341.408,A -85,B 0,C 180,E1 30374.392,E2 30374.392} C_VEL
LIN {X 0,Y 639.778,Z 341.532,A -85,B 0,C 180,E1 30373.703,E2 30373.703} C_VEL
LIN {X 0,Y 633.398,Z 342.325,A -85,B 0,C 180,E1 30371.771,E2 30371.771} C_VEL
LIN {X 0,Y 632.896,Z 342.388,A -85,B 0,C 180,E1 30371.269,E2 30371.269} C_VEL
LIN {X 0,Y 632.832,Z 342.397,A -85,B 0,C 180,E1 30368.254,E2 30368.254} C_VEL
LIN {X 0,Y 632.861,Z 342.391,A -85,B 0,C 180,E1 30365.387,E2 30365.387} C_VEL
LIN {X 0,Y 632.834,Z 342.397,A -85,B 0,C 180,E1 30362.172,E2 30362.172} C_VEL
LIN {X 0,Y 632.837,Z 342.392,A -85,B 0,C 180,E1 30359.431,E2 30359.431} C_VEL
LIN {X 0,Y 632.843,Z 342.396,A -85,B 0,C 180,E1 30356.156,E2 30356.156} C_VEL
LIN {X 0,Y 632.826,Z 342.39,A -85,B 0,C 180,E1 30353.363,E2 30353.363} C_VEL
LIN {X 0,Y 632.871,Z 342.394,A -85,B 0,C 180,E1 30350.243,E2 30350.243} C_VEL
LIN {X 0,Y 632.816,Z 342.398,A -85,B 0,C 180,E1 30347.375,E2 30347.375} C_VEL
LIN {X 0,Y 632.899,Z 342.391,A -85,B 0,C 180,E1 30344.361,E2 30344.361} C_VEL
LIN {X 0,Y 632.814,Z 342.402,A -85,B 0,C 180,E1 30341.391,E2 30341.391} C_VEL
LIN {X 0,Y 632.838,Z 342.4,A -85,B 0,C 180,E1 30338.633,E2 30338.633} C_VEL
LIN {X 0,Y 632.822,Z 342.397,A -85,B 0,C 180,E1 30335.44,E2 30335.44} C_VEL
LIN {X 0,Y 632.813,Z 342.398,A -85,B 0,C 180,E1 30332.717,E2 30332.717} C_VEL
LIN {X 0,Y 632.862,Z 342.4,A -85,B 0,C 180,E1 30329.638,E2 30329.638} C_VEL
LIN {X 0,Y 632.799,Z 342.38,A -85,B 0,C 180,E1 30326.83,E2 30326.83} C_VEL
LIN {X 0,Y 632.85,Z 342.387,A -85,B 0,C 180,E1 30324.015,E2 30324.015} C_VEL
LIN {X 0,Y 632.807,Z 342.405,A -85,B 0,C 180,E1 30320.909,E2 30320.909} C_VEL
LIN {X 0,Y 632.806,Z 342.391,A -85,B 0,C 180,E1 30318.239,E2 30318.239} C_VEL
LIN {X 0,Y 632.861,Z 342.539,A -85,B 0,C 180,E1 30315.801,E2 30315.801} C_VEL
LIN {X 0,Y 633.241,Z 343.96,A -85,B 0,C 180,E1 30315.6,E2 30315.6} C_VEL
LIN {X 0,Y 635.239,Z 347.08,A -85,B 0,C 180,E1 30315.32,E2 30315.32} C_VEL
LIN {X 0,Y 636.947,Z 348.75,A -85,B 0,C 180,E1 30315.105,E2 30315.105} C_VEL
LIN {X 0,Y 639.437,Z 352.557,A -85,B 0,C 180,E1 30314.77,E2 30314.77} C_VEL
LIN {X 0,Y 641.358,Z 354.799,A -85,B 0,C 180,E1 30314.527,E2 30314.527} C_VEL
LIN {X 0,Y 646.284,Z 361.521,A -85,B 0,C 180,E1 30313.9,E2 30313.9} C_VEL
LIN {X 0,Y 657.379,Z 376.504,A -85,B 0,C 180,E1 30312.564,E2 30312.564} C_VEL
LIN {X 0,Y 665.814,Z 388.548,A -85,B 0,C 180,E1 30311.597,E2 30311.597} C_VEL
LIN {X 0,Y 661.797,Z 606.523,A -85,B 0,C 180,E1 30308.669,E2 30308.669} C_VEL
LIN {X 0,Y 659.054,Z 757.476,A -85,B 0,C 180,E1 30306.667,E2 30306.667} C_VEL
LIN {X 0,Y 657.932,Z 783.583,A -85,B 0,C 180,E1 30306.175,E2 30306.175} C_VEL
LIN {X 0,Y 656.455,Z 810.606,A -85,B 0,C 180,E1 30305.495,E2 30305.495} C_VEL
LIN {X 0,Y 654.776,Z 836.686,A -85,B 0,C 180,E1 30304.665,E2 30304.665} C_VEL
LIN {X 0,Y 652.779,Z 863.3,A -85,B 0,C 180,E1 30303.628,E2 30303.628} C_VEL
LIN {X 0,Y 650.714,Z 887.709,A -85,B 0,C 180,E1 30302.495,E2 30302.495} C_VEL
LIN {X 0,Y 648.478,Z 912.743,A -85,B 0,C 180,E1 30301.14,E2 30301.14} C_VEL
LIN {X 0,Y 646.241,Z 936.376,A -85,B 0,C 180,E1 30299.663,E2 30299.663} C_VEL
LIN {X 0,Y 644.221,Z 956.959,A -85,B 0,C 180,E1 30298.202,E2 30298.202} C_VEL
LIN {X 0,Y 642.056,Z 979.099,A -85,B 0,C 180,E1 30296.426,E2 30296.426} C_VEL
LIN {X 0,Y 640.003,Z 1000.572,A -85,B 0,C 180,E1 30294.467,E2 30294.467} C_VEL
LIN {X 0,Y 638.138,Z 1020.483,A -85,B 0,C 180,E1 30292.41,E2 30292.41} C_VEL
LIN {X 0,Y 636.661,Z 1037.78,A -85,B 0,C 180,E1 30290.385,E2 30290.385} C_VEL
LIN {X 0,Y 635.347,Z 1054.069,A -85,B 0,C 180,E1 30288.243,E2 30288.243} C_VEL
LIN {X 0,Y 634.243,Z 1069.712,A -85,B 0,C 180,E1 30285.892,E2 30285.892} C_VEL
LIN {X 0,Y 633.497,Z 1081.758,A -85,B 0,C 180,E1 30283.838,E2 30283.838} C_VEL
LIN {X 0,Y 632.863,Z 1093.391,A -85,B 0,C 180,E1 30281.574,E2 30281.574} C_VEL
LIN {X 0,Y 632.434,Z 1104.246,A -85,B 0,C 180,E1 30279.08,E2 30279.08} C_VEL
LIN {X 0,Y 632.16,Z 1112.067,A -85,B 0,C 180,E1 30276.945,E2 30276.945} C_VEL
LIN {X 0,Y 632.029,Z 1119.122,A -85,B 0,C 180,E1 30274.608,E2 30274.608} C_VEL
LIN {X 0,Y 631.939,Z 1124.739,A -85,B 0,C 180,E1 30272.224,E2 30272.224} C_VEL
LIN {X 0,Y 631.923,Z 1128.637,A -85,B 0,C 180,E1 30269.878,E2 30269.878} C_VEL
LIN {X 0,Y 631.891,Z 1130.969,A -85,B 0,C 180,E1 30267.611,E2 30267.611} C_VEL
LIN {X 0,Y 631.899,Z 1131.916,A -85,B 0,C 180,E1 30265.393,E2 30265.393} C_VEL
LIN {X 0,Y 631.864,Z 1131.39,A -85,B 0,C 180,E1 30262.91,E2 30262.91} C_VEL
LIN {X 0,Y 631.916,Z 1129.352,A -85,B 0,C 180,E1 30260.565,E2 30260.565} C_VEL
LIN {X 0,Y 631.939,Z 1125.639,A -85,B 0,C 180,E1 30258.162,E2 30258.162} C_VEL
LIN {X 0,Y 632.005,Z 1120.165,A -85,B 0,C 180,E1 30255.696,E2 30255.696} C_VEL
LIN {X 0,Y 632.177,Z 1113.031,A -85,B 0,C 180,E1 30253.258,E2 30253.258} C_VEL
LIN {X 0,Y 632.394,Z 1105.377,A -85,B 0,C 180,E1 30251.122,E2 30251.122} C_VEL
LIN {X 0,Y 632.82,Z 1095.216,A -85,B 0,C 180,E1 30248.725,E2 30248.725} C_VEL
LIN {X 0,Y 633.413,Z 1083.242,A -85,B 0,C 180,E1 30246.344,E2 30246.344} C_VEL
LIN {X 0,Y 634.154,Z 1071.156,A -85,B 0,C 180,E1 30244.25,E2 30244.25} C_VEL
LIN {X 0,Y 635.192,Z 1056.314,A -85,B 0,C 180,E1 30241.985,E2 30241.985} C_VEL
LIN {X 0,Y 636.507,Z 1039.409,A -85,B 0,C 180,E1 30239.73,E2 30239.73} C_VEL
LIN {X 0,Y 637.945,Z 1022.764,A -85,B 0,C 180,E1 30237.754,E2 30237.754} C_VEL
LIN {X 0,Y 639.854,Z 1002.291,A -85,B 0,C 180,E1 30235.608,E2 30235.608} C_VEL
LIN {X 0,Y 641.781,Z 982.029,A -85,B 0,C 180,E1 30233.739,E2 30233.739} C_VEL
LIN {X 0,Y 644.047,Z 958.625,A -85,B 0,C 180,E1 30231.833,E2 30231.833} C_VEL
LIN {X 0,Y 646.316,Z 935.726,A -85,B 0,C 180,E1 30230.202,E2 30230.202} C_VEL
LIN {X 0,Y 648.579,Z 911.749,A -85,B 0,C 180,E1 30228.709,E2 30228.709} C_VEL
LIN {X 0,Y 650.745,Z 887.388,A -85,B 0,C 180,E1 30227.397,E2 30227.397} C_VEL
LIN {X 0,Y 652.801,Z 862.852,A -85,B 0,C 180,E1 30226.266,E2 30226.266} C_VEL
LIN {X 0,Y 654.722,Z 837.349,A -85,B 0,C 180,E1 30225.269,E2 30225.269} C_VEL
LIN {X 0,Y 656.349,Z 812.336,A -85,B 0,C 180,E1 30224.464,E2 30224.464} C_VEL
LIN {X 0,Y 657.859,Z 784.919,A -85,B 0,C 180,E1 30223.765,E2 30223.765} C_VEL
LIN {X 0,Y 658.994,Z 759.184,A -85,B 0,C 180,E1 30223.27,E2 30223.27} C_VEL
LIN {X 0,Y 660.271,Z 694.638,A -85,B 0,C 180,E1 30222.402,E2 30222.402} C_VEL
LIN {X 0,Y 664.297,Z 468.611,A -85,B 0,C 180,E1 30219.398,E2 30219.398} C_VEL
LIN {X 0,Y 665.737,Z 388.015,A -85,B 0,C 180,E1 30218.297,E2 30218.297} C_VEL
LIN {X 0,Y 650.619,Z 367.79,A -85,B 0,C 180,E1 30216.64,E2 30216.64} C_VEL
LIN {X 0,Y 643.637,Z 358.025,A -85,B 0,C 180,E1 30215.768,E2 30215.768} C_VEL
LIN {X 0,Y 640.388,Z 353.508,A -85,B 0,C 180,E1 30215.328,E2 30215.328} C_VEL
LIN {X 0,Y 637.63,Z 349.927,A -85,B 0,C 180,E1 30214.938,E2 30214.938} C_VEL
LIN {X 0,Y 636.615,Z 348.217,A -85,B 0,C 180,E1 30214.779,E2 30214.779} C_VEL
LIN {X 0,Y 634.023,Z 345.607,A -85,B 0,C 180,E1 30214.406,E2 30214.406} C_VEL
LIN {X 0,Y 632.986,Z 343,A -85,B 0,C 180,E1 30214.152,E2 30214.152} C_VEL
LIN {X 0,Y 632.864,Z 342.408,A -85,B 0,C 180,E1 30213.845,E2 30213.845} C_VEL
LIN {X 0,Y 632.871,Z 342.401,A -85,B 0,C 180,E1 30210.881,E2 30210.881} C_VEL
LIN {X 0,Y 632.868,Z 342.401,A -85,B 0,C 180,E1 30207.615,E2 30207.615} C_VEL
LIN {X 0,Y 632.915,Z 342.647,A -85,B 0,C 180,E1 30205.697,E2 30205.697} C_VEL
LIN {X 0,Y 634.298,Z 346.078,A -85,B 0,C 180,E1 30205.204,E2 30205.204} C_VEL
LIN {X 0,Y 638.392,Z 354.52,A -85,B 0,C 180,E1 30204.141,E2 30204.141} C_VEL
LIN {X 0,Y 644.033,Z 368.173,A -85,B 0,C 180,E1 30202.735,E2 30202.735} C_VEL
LIN {X 0,Y 650.296,Z 383.199,A -85,B 0,C 180,E1 30201.36,E2 30201.36} C_VEL
LIN {X 0,Y 657.152,Z 394.539,A -85,B 0,C 180,E1 30200.279,E2 30200.279} C_VEL
LIN {X 0,Y 657.556,Z 417.825,A -85,B 0,C 180,E1 30198.986,E2 30198.986} C_VEL
LIN {X 0,Y 661.722,Z 438.512,A -85,B 0,C 180,E1 30198.357,E2 30198.357} C_VEL
LIN {X 0,Y 666.769,Z 460.123,A -85,B 0,C 180,E1 30197.674,E2 30197.674} C_VEL
LIN {X 0,Y 665.393,Z 560.036,A -85,B 0,C 180,E1 30196.351,E2 30196.351} C_VEL
LIN {X 0,Y 661.412,Z 778.201,A -85,B 0,C 180,E1 30193.427,E2 30193.427} C_VEL
LIN {X 0,Y 659.068,Z 905.423,A -85,B 0,C 180,E1 30191.74,E2 30191.74} C_VEL
LIN {X 0,Y 658.006,Z 932.613,A -85,B 0,C 180,E1 30191.243,E2 30191.243} C_VEL
LIN {X 0,Y 656.57,Z 958.486,A -85,B 0,C 180,E1 30190.598,E2 30190.598} C_VEL
LIN {X 0,Y 655.164,Z 980.371,A -85,B 0,C 180,E1 30189.922,E2 30189.922} C_VEL
LIN {X 0,Y 653.723,Z 1000.863,A -85,B 0,C 180,E1 30189.175,E2 30189.175} C_VEL
LIN {X 0,Y 651.888,Z 1024.345,A -85,B 0,C 180,E1 30188.179,E2 30188.179} C_VEL
LIN {X 0,Y 649.628,Z 1050.14,A -85,B 0,C 180,E1 30186.889,E2 30186.889} C_VEL
LIN {X 0,Y 647.699,Z 1070.818,A -85,B 0,C 180,E1 30185.699,E2 30185.699} C_VEL
LIN {X 0,Y 645.792,Z 1090.733,A -85,B 0,C 180,E1 30184.411,E2 30184.411} C_VEL
LIN {X 0,Y 643.562,Z 1113.754,A -85,B 0,C 180,E1 30182.729,E2 30182.729} C_VEL
LIN {X 0,Y 641.583,Z 1133.832,A -85,B 0,C 180,E1 30181.054,E2 30181.054} C_VEL
LIN {X 0,Y 640.007,Z 1150.448,A -85,B 0,C 180,E1 30179.517,E2 30179.517} C_VEL
LIN {X 0,Y 638.37,Z 1168.009,A -85,B 0,C 180,E1 30177.722,E2 30177.722} C_VEL
LIN {X 0,Y 636.766,Z 1186.521,A -85,B 0,C 180,E1 30175.583,E2 30175.583} C_VEL
LIN {X 0,Y 635.535,Z 1201.395,A -85,B 0,C 180,E1 30173.652,E2 30173.652} C_VEL
LIN {X 0,Y 634.498,Z 1215.919,A -85,B 0,C 180,E1 30171.541,E2 30171.541} C_VEL
LIN {X 0,Y 633.592,Z 1230.191,A -85,B 0,C 180,E1 30169.162,E2 30169.162} C_VEL
LIN {X 0,Y 632.986,Z 1241.078,A -85,B 0,C 180,E1 30167.086,E2 30167.086} C_VEL
LIN {X 0,Y 632.584,Z 1250.525,A -85,B 0,C 180,E1 30165.024,E2 30165.024} C_VEL
LIN {X 0,Y 632.234,Z 1260.302,A -85,B 0,C 180,E1 30162.513,E2 30162.513} C_VEL
LIN {X 0,Y 632.068,Z 1267.354,A -85,B 0,C 180,E1 30160.273,E2 30160.273} C_VEL
LIN {X 0,Y 631.955,Z 1272.943,A -85,B 0,C 180,E1 30158.095,E2 30158.095} C_VEL
LIN {X 0,Y 631.931,Z 1277.337,A -85,B 0,C 180,E1 30155.812,E2 30155.812} C_VEL
LIN {X 0,Y 631.909,Z 1280.404,A -85,B 0,C 180,E1 30153.356,E2 30153.356} C_VEL
LIN {X 0,Y 631.888,Z 1281.714,A -85,B 0,C 180,E1 30151.179,E2 30151.179} C_VEL
LIN {X 0,Y 631.863,Z 1281.827,A -85,B 0,C 180,E1 30149.275,E2 30149.275} C_VEL
LIN {X 0,Y 631.907,Z 1280.947,A -85,B 0,C 180,E1 30147.37,E2 30147.37} C_VEL
LIN {X 0,Y 631.914,Z 1278.901,A -85,B 0,C 180,E1 30145.28,E2 30145.28} C_VEL
LIN {X 0,Y 631.951,Z 1275.078,A -85,B 0,C 180,E1 30142.911,E2 30142.911} C_VEL
LIN {X 0,Y 631.973,Z 1269.838,A -85,B 0,C 180,E1 30140.621,E2 30140.621} C_VEL
LIN {X 0,Y 632.154,Z 1263.356,A -85,B 0,C 180,E1 30138.412,E2 30138.412} C_VEL
LIN {X 0,Y 632.323,Z 1256.515,A -85,B 0,C 180,E1 30136.466,E2 30136.466} C_VEL
LIN {X 0,Y 632.645,Z 1248.489,A -85,B 0,C 180,E1 30134.508,E2 30134.508} C_VEL
LIN {X 0,Y 633.137,Z 1238.287,A -85,B 0,C 180,E1 30132.349,E2 30132.349} C_VEL
LIN {X 0,Y 633.917,Z 1224.733,A -85,B 0,C 180,E1 30129.888,E2 30129.888} C_VEL
LIN {X 0,Y 634.783,Z 1211.882,A -85,B 0,C 180,E1 30127.851,E2 30127.851} C_VEL
LIN {X 0,Y 635.901,Z 1197.144,A -85,B 0,C 180,E1 30125.771,E2 30125.771} C_VEL
LIN {X 0,Y 637.366,Z 1179.224,A -85,B 0,C 180,E1 30123.543,E2 30123.543} C_VEL
LIN {X 0,Y 638.835,Z 1162.917,A -85,B 0,C 180,E1 30121.741,E2 30121.741} C_VEL
LIN {X 0,Y 640.483,Z 1145.389,A -85,B 0,C 180,E1 30119.994,E2 30119.994} C_VEL
LIN {X 0,Y 642.597,Z 1123.475,A -85,B 0,C 180,E1 30118.06,E2 30118.06} C_VEL
LIN {X 0,Y 644.434,Z 1104.718,A -85,B 0,C 180,E1 30116.59,E2 30116.59} C_VEL
LIN {X 0,Y 646.228,Z 1086.318,A -85,B 0,C 180,E1 30115.292,E2 30115.292} C_VEL
LIN {X 0,Y 648.432,Z 1063.509,A -85,B 0,C 180,E1 30113.856,E2 30113.856} C_VEL
LIN {X 0,Y 650.61,Z 1038.71,A -85,B 0,C 180,E1 30112.513,E2 30112.513} C_VEL
LIN {X 0,Y 652.377,Z 1017.593,A -85,B 0,C 180,E1 30111.518,E2 30111.518} C_VEL
LIN {X 0,Y 654.076,Z 995.723,A -85,B 0,C 180,E1 30110.624,E2 30110.624} C_VEL
LIN {X 0,Y 656.019,Z 968.196,A -85,B 0,C 180,E1 30109.682,E2 30109.682} C_VEL
LIN {X 0,Y 657.422,Z 943.256,A -85,B 0,C 180,E1 30109.006,E2 30109.006} C_VEL
LIN {X 0,Y 658.501,Z 920.428,A -85,B 0,C 180,E1 30108.516,E2 30108.516} C_VEL
LIN {X 0,Y 659.404,Z 894.503,A -85,B 0,C 180,E1 30108.1,E2 30108.1} C_VEL
LIN {X 0,Y 663.338,Z 670.296,A -85,B 0,C 180,E1 30105.137,E2 30105.137} C_VEL
LIN {X 0,Y 666.892,Z 474.641,A -85,B 0,C 180,E1 30102.49,E2 30102.49} C_VEL
LIN {X 0,Y 666.993,Z 458.644,A -85,B 0,C 180,E1 30102.256,E2 30102.256} C_VEL
LIN {X 0,Y 659.903,Z 424.22,A -85,B 0,C 180,E1 30101.013,E2 30101.013} C_VEL
LIN {X 0,Y 661.188,Z 397.914,A -85,B 0,C 180,E1 30099.288,E2 30099.288} C_VEL
LIN {X 0,Y 648.683,Z 372.947,A -85,B 0,C 180,E1 30096.183,E2 30096.183} C_VEL
LIN {X 0,Y 642.339,Z 360.688,A -85,B 0,C 180,E1 30094.515,E2 30094.515} C_VEL
LIN {X 0,Y 637.457,Z 351.506,A -85,B 0,C 180,E1 30093.191,E2 30093.191} C_VEL
LIN {X 0,Y 634.887,Z 346.798,A -85,B 0,C 180,E1 30092.483,E2 30092.483} C_VEL
LIN {X 0,Y 633.058,Z 343.313,A -85,B 0,C 180,E1 30091.946,E2 30091.946} C_VEL
LIN {X 0,Y 632.895,Z 342.495,A -85,B 0,C 180,E1 30091.742,E2 30091.742} C_VEL
LIN {X 0,Y 632.871,Z 342.388,A -85,B 0,C 180,E1 30088.705,E2 30088.705} C_VEL
LIN {X 0,Y 632.883,Z 342.391,A -85,B 0,C 180,E1 30085.563,E2 30085.563} C_VEL
LIN {X 0,Y 632.866,Z 342.4,A -85,B 0,C 180,E1 30082.444,E2 30082.444} C_VEL
LIN {X 0,Y 632.886,Z 342.396,A -85,B 0,C 180,E1 30079.377,E2 30079.377} C_VEL
LIN {X 0,Y 632.862,Z 342.396,A -85,B 0,C 180,E1 30076.239,E2 30076.239} C_VEL
LIN {X 0,Y 632.886,Z 342.396,A -85,B 0,C 180,E1 30073.15,E2 30073.15} C_VEL
LIN {X 0,Y 632.859,Z 342.396,A -85,B 0,C 180,E1 30070.009,E2 30070.009} C_VEL
LIN {X 0,Y 632.887,Z 342.394,A -85,B 0,C 180,E1 30066.987,E2 30066.987} C_VEL
LIN {X 0,Y 632.858,Z 342.399,A -85,B 0,C 180,E1 30063.896,E2 30063.896} C_VEL
LIN {X 0,Y 632.888,Z 342.385,A -85,B 0,C 180,E1 30060.815,E2 30060.815} C_VEL
LIN {X 0,Y 632.856,Z 342.397,A -85,B 0,C 180,E1 30057.736,E2 30057.736} C_VEL
LIN {X 0,Y 632.89,Z 342.391,A -85,B 0,C 180,E1 30054.651,E2 30054.651} C_VEL
LIN {X 0,Y 632.852,Z 342.397,A -85,B 0,C 180,E1 30051.55,E2 30051.55} C_VEL
LIN {X 0,Y 632.89,Z 342.392,A -85,B 0,C 180,E1 30048.518,E2 30048.518} C_VEL
LIN {X 0,Y 632.853,Z 342.398,A -85,B 0,C 180,E1 30045.45,E2 30045.45} C_VEL
LIN {X 0,Y 632.886,Z 342.385,A -85,B 0,C 180,E1 30042.437,E2 30042.437} C_VEL
LIN {X 0,Y 632.852,Z 342.398,A -85,B 0,C 180,E1 30039.273,E2 30039.273} C_VEL
LIN {X 0,Y 632.886,Z 342.385,A -85,B 0,C 180,E1 30036.242,E2 30036.242} C_VEL
LIN {X 0,Y 632.847,Z 342.398,A -85,B 0,C 180,E1 30033.034,E2 30033.034} C_VEL
LIN {X 0,Y 632.887,Z 342.386,A -85,B 0,C 180,E1 30030.05,E2 30030.05} C_VEL
LIN {X 0,Y 632.844,Z 342.398,A -85,B 0,C 180,E1 30026.86,E2 30026.86} C_VEL
LIN {X 0,Y 632.878,Z 342.388,A -85,B 0,C 180,E1 30023.892,E2 30023.892} C_VEL
LIN {X 0,Y 632.844,Z 342.398,A -85,B 0,C 180,E1 30020.731,E2 30020.731} C_VEL
LIN {X 0,Y 632.862,Z 342.39,A -85,B 0,C 180,E1 30017.818,E2 30017.818} C_VEL
LIN {X 0,Y 632.85,Z 342.396,A -85,B 0,C 180,E1 30014.675,E2 30014.675} C_VEL
LIN {X 0,Y 632.842,Z 342.392,A -85,B 0,C 180,E1 30011.817,E2 30011.817} C_VEL
LIN {X 0,Y 632.896,Z 342.388,A -85,B 0,C 180,E1 30011.269,E2 30011.269} C_VEL
LIN {X 0,Y 631.931,Z 342.515,A -85,B 0,C 180,E1 30010.572,E2 30010.572} C_VEL
LIN {X 0,Y 625.433,Z 343.321,A -85,B 0,C 180,E1 30008.617,E2 30008.617} C_VEL
LIN {X 0,Y 624.889,Z 343.386,A -85,B 0,C 180,E1 30008.108,E2 30008.108} C_VEL
LIN {X 0,Y 624.953,Z 343.378,A -85,B 0,C 180,E1 30005.056,E2 30005.056} C_VEL
LIN {X 0,Y 624.887,Z 343.386,A -85,B 0,C 180,E1 30001.98,E2 30001.98} C_VEL
LIN {X 0,Y 624.931,Z 343.378,A -85,B 0,C 180,E1 29999.104,E2 29999.104} C_VEL
LIN {X 0,Y 624.889,Z 343.387,A -85,B 0,C 180,E1 29995.938,E2 29995.938} C_VEL
LIN {X 0,Y 624.908,Z 343.377,A -85,B 0,C 180,E1 29993.08,E2 29993.08} C_VEL
LIN {X 0,Y 624.89,Z 343.39,A -85,B 0,C 180,E1 29989.829,E2 29989.829} C_VEL
LIN {X 0,Y 624.893,Z 343.385,A -85,B 0,C 180,E1 29987.026,E2 29987.026} C_VEL
LIN {X 0,Y 624.892,Z 343.39,A -85,B 0,C 180,E1 29983.698,E2 29983.698} C_VEL
LIN {X 0,Y 624.88,Z 343.39,A -85,B 0,C 180,E1 29980.977,E2 29980.977} C_VEL
LIN {X 0,Y 624.916,Z 343.385,A -85,B 0,C 180,E1 29977.817,E2 29977.817} C_VEL
LIN {X 0,Y 624.868,Z 343.384,A -85,B 0,C 180,E1 29975.049,E2 29975.049} C_VEL
LIN {X 0,Y 624.945,Z 343.382,A -85,B 0,C 180,E1 29972.017,E2 29972.017} C_VEL
LIN {X 0,Y 624.871,Z 343.393,A -85,B 0,C 180,E1 29969.083,E2 29969.083} C_VEL
LIN {X 0,Y 624.883,Z 343.37,A -85,B 0,C 180,E1 29966.33,E2 29966.33} C_VEL
LIN {X 0,Y 624.876,Z 343.366,A -85,B 0,C 180,E1 29963.107,E2 29963.107} C_VEL
LIN {X 0,Y 624.864,Z 343.385,A -85,B 0,C 180,E1 29960.421,E2 29960.421} C_VEL
LIN {X 0,Y 624.924,Z 343.386,A -85,B 0,C 180,E1 29957.338,E2 29957.338} C_VEL
LIN {X 0,Y 624.891,Z 343.598,A -85,B 0,C 180,E1 29956.679,E2 29956.679} C_VEL
LIN {X 0,Y 625.262,Z 345.068,A -85,B 0,C 180,E1 29956.481,E2 29956.481} C_VEL
LIN {X 0,Y 627.083,Z 347.95,A -85,B 0,C 180,E1 29956.214,E2 29956.214} C_VEL
LIN {X 0,Y 629.19,Z 349.844,A -85,B 0,C 180,E1 29955.94,E2 29955.94} C_VEL
LIN {X 0,Y 631.88,Z 353.813,A -85,B 0,C 180,E1 29955.567,E2 29955.567} C_VEL
LIN {X 0,Y 633.461,Z 355.712,A -85,B 0,C 180,E1 29955.358,E2 29955.358} C_VEL
LIN {X 0,Y 636.834,Z 360.072,A -85,B 0,C 180,E1 29954.913,E2 29954.913} C_VEL
LIN {X 0,Y 652.795,Z 381.78,A -85,B 0,C 180,E1 29952.918,E2 29952.918} C_VEL
LIN {X 0,Y 660.213,Z 392.47,A -85,B 0,C 180,E1 29952.049,E2 29952.049} C_VEL
LIN {X 0,Y 655.953,Z 609.718,A -85,B 0,C 180,E1 29949.111,E2 29949.111} C_VEL
LIN {X 0,Y 653.074,Z 757.561,A -85,B 0,C 180,E1 29947.135,E2 29947.135} C_VEL
LIN {X 0,Y 651.879,Z 783.767,A -85,B 0,C 180,E1 29946.638,E2 29946.638} C_VEL
LIN {X 0,Y 650.315,Z 810.707,A -85,B 0,C 180,E1 29945.956,E2 29945.956} C_VEL
LIN {X 0,Y 648.55,Z 836.421,A -85,B 0,C 180,E1 29945.134,E2 29945.134} C_VEL
LIN {X 0,Y 646.558,Z 861.833,A -85,B 0,C 180,E1 29944.145,E2 29944.145} C_VEL
LIN {X 0,Y 644.271,Z 886.963,A -85,B 0,C 180,E1 29942.979,E2 29942.979} C_VEL
LIN {X 0,Y 641.884,Z 911.794,A -85,B 0,C 180,E1 29941.634,E2 29941.634} C_VEL
LIN {X 0,Y 639.479,Z 935.731,A -85,B 0,C 180,E1 29940.132,E2 29940.132} C_VEL
LIN {X 0,Y 637.327,Z 956.308,A -85,B 0,C 180,E1 29938.663,E2 29938.663} C_VEL
LIN {X 0,Y 634.983,Z 978.424,A -85,B 0,C 180,E1 29936.879,E2 29936.879} C_VEL
LIN {X 0,Y 632.794,Z 999.618,A -85,B 0,C 180,E1 29934.936,E2 29934.936} C_VEL
LIN {X 0,Y 630.808,Z 1019.502,A -85,B 0,C 180,E1 29932.874,E2 29932.874} C_VEL
LIN {X 0,Y 629.101,Z 1037.746,A -85,B 0,C 180,E1 29930.718,E2 29930.718} C_VEL
LIN {X 0,Y 627.63,Z 1054.495,A -85,B 0,C 180,E1 29928.484,E2 29928.484} C_VEL
LIN {X 0,Y 626.454,Z 1069.768,A -85,B 0,C 180,E1 29926.156,E2 29926.156} C_VEL
LIN {X 0,Y 625.626,Z 1082.151,A -85,B 0,C 180,E1 29924.012,E2 29924.012} C_VEL
LIN {X 0,Y 624.943,Z 1093.681,A -85,B 0,C 180,E1 29921.728,E2 29921.728} C_VEL
LIN {X 0,Y 624.479,Z 1104.49,A -85,B 0,C 180,E1 29919.2,E2 29919.2} C_VEL
LIN {X 0,Y 624.179,Z 1112.278,A -85,B 0,C 180,E1 29917.037,E2 29917.037} C_VEL
LIN {X 0,Y 624.037,Z 1119.293,A -85,B 0,C 180,E1 29914.668,E2 29914.668} C_VEL
LIN {X 0,Y 623.939,Z 1124.859,A -85,B 0,C 180,E1 29912.252,E2 29912.252} C_VEL
LIN {X 0,Y 623.924,Z 1128.706,A -85,B 0,C 180,E1 29909.89,E2 29909.89} C_VEL
LIN {X 0,Y 623.89,Z 1131.01,A -85,B 0,C 180,E1 29907.592,E2 29907.592} C_VEL
LIN {X 0,Y 623.899,Z 1131.93,A -85,B 0,C 180,E1 29905.327,E2 29905.327} C_VEL
LIN {X 0,Y 623.864,Z 1131.352,A -85,B 0,C 180,E1 29902.822,E2 29902.822} C_VEL
LIN {X 0,Y 623.916,Z 1129.394,A -85,B 0,C 180,E1 29900.547,E2 29900.547} C_VEL
LIN {X 0,Y 623.941,Z 1125.761,A -85,B 0,C 180,E1 29898.142,E2 29898.142} C_VEL
LIN {X 0,Y 624.016,Z 1120.264,A -85,B 0,C 180,E1 29895.616,E2 29895.616} C_VEL
LIN {X 0,Y 624.193,Z 1113.17,A -85,B 0,C 180,E1 29893.148,E2 29893.148} C_VEL
LIN {X 0,Y 624.44,Z 1105.54,A -85,B 0,C 180,E1 29890.985,E2 29890.985} C_VEL
LIN {X 0,Y 624.894,Z 1095.42,A -85,B 0,C 180,E1 29888.558,E2 29888.558} C_VEL
LIN {X 0,Y 625.545,Z 1083.496,A -85,B 0,C 180,E1 29886.148,E2 29886.148} C_VEL
LIN {X 0,Y 626.348,Z 1071.444,A -85,B 0,C 180,E1 29884.028,E2 29884.028} C_VEL
LIN {X 0,Y 627.467,Z 1056.648,A -85,B 0,C 180,E1 29881.735,E2 29881.735} C_VEL
LIN {X 0,Y 628.9,Z 1039.8,A -85,B 0,C 180,E1 29879.453,E2 29879.453} C_VEL
LIN {X 0,Y 630.432,Z 1023.199,A -85,B 0,C 180,E1 29877.455,E2 29877.455} C_VEL
LIN {X 0,Y 632.493,Z 1002.798,A -85,B 0,C 180,E1 29875.285,E2 29875.285} C_VEL
LIN {X 0,Y 634.558,Z 982.578,A -85,B 0,C 180,E1 29873.395,E2 29873.395} C_VEL
LIN {X 0,Y 637.004,Z 959.233,A -85,B 0,C 180,E1 29871.47,E2 29871.47} C_VEL
LIN {X 0,Y 639.421,Z 936.413,A -85,B 0,C 180,E1 29869.822,E2 29869.822} C_VEL
LIN {X 0,Y 641.842,Z 912.531,A -85,B 0,C 180,E1 29868.316,E2 29868.316} C_VEL
LIN {X 0,Y 644.156,Z 888.212,A -85,B 0,C 180,E1 29866.993,E2 29866.993} C_VEL
LIN {X 0,Y 646.351,Z 863.778,A -85,B 0,C 180,E1 29865.852,E2 29865.852} C_VEL
LIN {X 0,Y 648.403,Z 838.461,A -85,B 0,C 180,E1 29864.848,E2 29864.848} C_VEL
LIN {X 0,Y 650.158,Z 813.008,A -85,B 0,C 180,E1 29864.021,E2 29864.021} C_VEL
LIN {X 0,Y 651.776,Z 785.63,A -85,B 0,C 180,E1 29863.315,E2 29863.315} C_VEL
LIN {X 0,Y 652.967,Z 760.193,A -85,B 0,C 180,E1 29862.819,E2 29862.819} C_VEL
LIN {X 0,Y 654.076,Z 710.997,A -85,B 0,C 180,E1 29862.143,E2 29862.143} C_VEL
LIN {X 0,Y 658.344,Z 486.34,A -85,B 0,C 180,E1 29859.14,E2 29859.14} C_VEL
LIN {X 0,Y 659.856,Z 391.884,A -85,B 0,C 180,E1 29857.856,E2 29857.856} C_VEL
LIN {X 0,Y 646.764,Z 374.115,A -85,B 0,C 180,E1 29856.373,E2 29856.373} C_VEL
LIN {X 0,Y 639.3,Z 363.632,A -85,B 0,C 180,E1 29855.408,E2 29855.408} C_VEL
LIN {X 0,Y 636.488,Z 359.747,A -85,B 0,C 180,E1 29855.016,E2 29855.016} C_VEL
LIN {X 0,Y 633.487,Z 355.305,A -85,B 0,C 180,E1 29854.555,E2 29854.555} C_VEL
LIN {X 0,Y 630.454,Z 351.839,A -85,B 0,C 180,E1 29854.087,E2 29854.087} C_VEL
LIN {X 0,Y 629.264,Z 349.56,A -85,B 0,C 180,E1 29853.865,E2 29853.865} C_VEL
